FUNCTION_BLOCK TaskStoppingProbe EXTENDS TOF_Tasks.Task
VAR_INPUT
	//! <summary>Ordinary OnRunning result when no exception is injected.</summary>
	ProcessingResult : TOF_Tasks.TASK_PROCESSING_STATE := TOF_Tasks.TASK_PROCESSING_STATE.DONE;
	//! <summary>Throw from start preparation before RUNNING is entered.</summary>
	ThrowOnBeforeStart : BOOL;
	//! <summary>Throw when ordinary processing is called.</summary>
	ThrowOnRunning : BOOL;
	//! <summary>Throw once in stopping before advancing cleanup.</summary>
	ThrowOnFirstStopping : BOOL;
	//! <summary>Throw on every stopping call while enabled, before advancing cleanup.</summary>
	ThrowOnEveryStopping : BOOL;
	//! <summary>Throw from reset before descendant state is cleared.</summary>
	ThrowOnReset : BOOL;
	//! <summary>Injected exceptions throw again from GetMessage.</summary>
	ThrowOnGetMessage : BOOL;
	//! <summary>Throw a StandardException whose GetMessage result is empty.</summary>
	ThrowWithEmptyMessage : BOOL;
	//! <summary>Exercise the permitted Reset notification after termination.</summary>
	ResetOnAfterStop : BOOL;
END_VAR
VAR_OUTPUT
	//! <summary>Total ordinary processing calls across runs.</summary>
	RunningCalls : UINT;
	//! <summary>Total stopping-hook calls across runs, including interrupted calls.</summary>
	StoppingCalls : UINT;
	//! <summary>Successful stopping steps since the last Reset.</summary>
	CompletedCleanupSteps : UINT;
	//! <summary>Total notifications after STOPPED has been recorded.</summary>
	AfterStopCalls : UINT;
	//! <summary>Total accepted cancellation notifications.</summary>
	CancelNotifications : UINT;
END_VAR
VAR CONSTANT
	//! <summary>Successful cleanup steps required before release is safe.</summary>
	_CleanupSteps : UINT := 2;
END_VAR
VAR_STAT
	//! <summary>Class name shared by all instances of this function block.</summary>
	_ClassName : STRING := __POUNAME();
END_VAR
VAR
	_Resource : REFERENCE TO TaskStoppingResource;
	_StoppingExceptionRaised : BOOL;
END_VAR

{attribute 'monitoring' := 'call'}
PROPERTY ClassName : REFERENCE TO STRING
GET
ClassName REF= _ClassName;
END_GET
END_PROPERTY

(*!
<summary>Starts a fresh set of observation counts.</summary>
<description>
Call while the fixture is READY. Leaves configuration, cleanup progress and the borrowed resource binding intact.
</description>
*)
METHOD INTERNAL ClearObservations
RunningCalls := 0;
StoppingCalls := 0;
AfterStopCalls := 0;
CancelNotifications := 0;
END_METHOD

(*!
<summary>Borrows the test namespace.</summary>
*)
{attribute 'monitoring' := 'call'}
PROPERTY NamespaceName : REFERENCE TO STRING
GET
NamespaceName REF= CurrentNamespace.Name;
END_GET
END_PROPERTY

(*!
<summary>Counts finalization and optionally resets the stopped task.</summary>
<description>
Reset is invoked only after STOPPED and final diagnostics have been published.
</description>
*)
METHOD PROTECTED OnAfterStop
AfterStopCalls := AfterStopCalls + 1;

IF ResetOnAfterStop THEN
	Reset();
END_IF
END_METHOD

(*!
<summary>Optionally refuses start through an injected exception.</summary>
*)
METHOD PROTECTED OnBeforeStart
IF ThrowOnBeforeStart THEN
	raiseConfiguredFailure(message := "Start failure");
END_IF
END_METHOD

(*!
<summary>Counts accepted external cancellation notifications.</summary>
*)
METHOD PROTECTED OnCancelRequest
CancelNotifications := CancelNotifications + 1;
END_METHOD

(*!
<summary>Clears per-run cleanup progress without resetting observations or the dependency.</summary>
<description>
An injected exception refuses Reset before changing descendant state.
</description>
*)
METHOD PROTECTED OnReset
IF ThrowOnReset THEN
	raiseConfiguredFailure(message := "Reset failure");
END_IF

CompletedCleanupSteps := 0;
_StoppingExceptionRaised := FALSE;
END_METHOD

(*!
<summary>Returns the configured work result or injects a processing exception.</summary>
<description>
One call records one unit of work; no resource operations are driven here.
</description>
<param name="processingState">Configured result on normal return.</param>
<param name="stopReasonMessage">Receives diagnostic text for ERROR or ABORTED.</param>
*)
METHOD PROTECTED OnRunning
VAR_OUTPUT
	processingState : TOF_Tasks.TASK_PROCESSING_STATE;
END_VAR
VAR_IN_OUT
	stopReasonMessage : TOF_Core.ERROR_MESSAGE;
END_VAR
RunningCalls := RunningCalls + 1;

IF ThrowOnRunning THEN
	raiseConfiguredFailure(message := "Work failure");
END_IF

processingState := ProcessingResult;

IF processingState = TOF_Tasks.TASK_PROCESSING_STATE.ERROR
	OR_ELSE processingState = TOF_Tasks.TASK_PROCESSING_STATE.ABORTED
THEN
	stopReasonMessage := "Work result";
END_IF
END_METHOD

(*!
<summary>Finishes late acquisition and two cleanup steps before allowing release.</summary>
<description>
The configured exception can interrupt one or every call before progress. A later call resumes without
rerunning ordinary work once repeated injection is disabled.
</description>
<param name="readyToRelease">TRUE only after pending acquisition and cleanup have completed.</param>
*)
METHOD PROTECTED OnStopping
VAR_OUTPUT
	readyToRelease : BOOL;
END_VAR
StoppingCalls := StoppingCalls + 1;

IF ThrowOnFirstStopping AND_THEN NOT _StoppingExceptionRaised THEN
	_StoppingExceptionRaised := TRUE;
	raiseConfiguredFailure(message := "Stopping failure");
END_IF

IF ThrowOnEveryStopping THEN
	raiseConfiguredFailure(message := "Stopping failure");
END_IF

IF __ISVALIDREF(_Resource) AND_THEN NOT _Resource.FinishPendingAcquire() THEN
	RETURN;
END_IF

CompletedCleanupSteps := CompletedCleanupSteps + 1;
readyToRelease := CompletedCleanupSteps >= _CleanupSteps;
END_METHOD

(*!
<summary>Raises the configured synthetic exception.</summary>
<description>
Used only by test operations, never by FB lifecycle methods. A throwing or empty formatter exercises
diagnostic fallback.
</description>
<param name="message">Text copied into the injected exception.</param>
*)
METHOD PRIVATE raiseConfiguredFailure
VAR_INPUT
	message : WSTRING(255);
END_VAR
VAR
	failure : TOF_Core.StandardException;
	formattingFailure : ThrowingGetMessageException;
	emptyMessage : TOF_Core.ERROR_MESSAGE;
END_VAR
IF ThrowOnGetMessage THEN
	formattingFailure.Throw(
		sourceNamespaceName := NamespaceName,
		sourceClassName := ClassName,
		sourcePOUName := __POUNAME(),
		sourcePosition := __POSITION(),
		message := message
	);
ELSIF ThrowWithEmptyMessage THEN
	emptyMessage := TOF_Core.WideStrings.Empty;
	failure.Throw(
		sourceNamespaceName := NamespaceName,
		sourceClassName := ClassName,
		sourcePOUName := __POUNAME(),
		sourcePosition := __POSITION(),
		message := emptyMessage
	);
ELSE
	failure.Throw(
		sourceNamespaceName := NamespaceName,
		sourceClassName := ClassName,
		sourcePOUName := __POUNAME(),
		sourcePosition := __POSITION(),
		message := message
	);
END_IF
END_METHOD

(*!
<summary>Returns the explicitly injected borrowed resource manager.</summary>
<description>
Zero before binding; getter has no side effects and does not throw.
</description>
*)
{attribute 'monitoring' := 'call'}
PROPERTY ResourceManager : TOF_Core.IResourceManager
GET
IF __ISVALIDREF(_Resource) THEN
	ResourceManager := _Resource;
END_IF
END_GET
END_PROPERTY

(*!
<summary>Reports the concrete fixture size.</summary>
*)
{attribute 'monitoring' := 'call'}
PROPERTY SelfSize : ULINT
GET
SelfSize := XSIZEOF(THIS^);
END_GET
END_PROPERTY

(*!
<summary>Binds the manager owned by the scenario.</summary>
<description>
Call before Start and keep the referenced manager alive and unchanged throughout every run. Reset preserves
the binding.
</description>
<param name="resource">Live synthetic manager owned directly by the scenario.</param>
*)
METHOD INTERNAL SetResource
VAR_IN_OUT
	resource : TaskStoppingResource;
END_VAR
_Resource REF= resource;
END_METHOD

END_FUNCTION_BLOCK

// ---- Tests/Tasks/Stopping/TaskStoppingResource.TcPOU
(*
SPDX-FileCopyrightText: © 2026 Oleksandr Tiutyk <trofimich@gmail.com>
SPDX-License-Identifier: MIT
License: https://opensource.org/license/mit
*)

(*!
<summary>Provides delayed synthetic acquisition and release for Task stopping tests.</summary>
<description>
The scenario owns this manager and injects it into the task explicitly. Configure inputs before Start.
Operations have no hardware effects. A release exception intentionally leaves the synthetic resource held.
Observations are read-only to the scenario. ResetFixture clears them and the simulated state once the task is inactive.
</description>
*)

FUNCTION_BLOCK TaskStoppingResource EXTENDS TOF_Core.Object IMPLEMENTS TOF_Core.IResourceManager
VAR_INPUT
	//! <summary>Throw before acquisition is scheduled.</summary>
	ThrowOnStartAcquire : BOOL;
	//! <summary>Throw after the last acquisition step has marked the resource acquired.</summary>
	ThrowAfterAcquire : BOOL;
	//! <summary>Throw before release is scheduled, retaining the acquired resource.</summary>
	ThrowOnStartRelease : BOOL;
	//! <summary>Injected exceptions throw again when GetMessage is called.</summary>
	ThrowOnGetMessage : BOOL;
END_VAR
VAR_OUTPUT
	//! <summary>Total acquisition requests across runs.</summary>
	AcquireCalls : UINT;
	//! <summary>Total release requests across runs.</summary>
	ReleaseCalls : UINT;
	//! <summary>Completed steps in the current acquisition.</summary>
	AcquireProgress : UINT;
END_VAR
VAR CONSTANT
	//! <summary>Calls needed for a pending acquisition, allowing cancellation before its response.</summary>
	_AcquireSteps : UINT := 3;
	//! <summary>Calls needed after StartRelease to observe asynchronous completion.</summary>
	_ReleaseSteps : UINT := 2;
END_VAR
VAR_STAT
	//! <summary>Class name shared by all instances of this function block.</summary>
	_ClassName : STRING := __POUNAME();
END_VAR
VAR
	_Acquired : BOOL;
	_Acquiring : BOOL;
	_Releasing : BOOL;
	_ReleaseProgress : UINT;
END_VAR

{attribute 'monitoring' := 'call'}
PROPERTY ClassName : REFERENCE TO STRING
GET
ClassName REF= _ClassName;
END_GET
END_PROPERTY

(*!
<summary>Advances one pending synthetic operation.</summary>
<description>
No pending operation means no action. Acquisition failure may occur after ownership was obtained.
</description>
*)
METHOD Execute
IF _Acquiring THEN
	AcquireProgress := AcquireProgress + 1;

	IF AcquireProgress >= _AcquireSteps THEN
		_Acquiring := FALSE;
		_Acquired := TRUE;

		IF ThrowAfterAcquire THEN
			raiseConfiguredFailure(message := "Acquire failure");
		END_IF
	END_IF
ELSIF _Releasing THEN
	_ReleaseProgress := _ReleaseProgress + 1;

	IF _ReleaseProgress >= _ReleaseSteps THEN
		_Releasing := FALSE;
		_Acquired := FALSE;
	END_IF
END_IF
END_METHOD

(*!
<summary>Drains a late acquisition response without starting a new request.</summary>
<description>
Used by the injected task during OnStopping. A late acquired resource remains available for normal release.
</description>
*)
METHOD INTERNAL FinishPendingAcquire : BOOL
IF _Acquiring THEN
	Execute();
END_IF

FinishPendingAcquire := NOT _Acquiring;
END_METHOD

(*!
<summary>Returns the borrowed manager as a synthetic resource.</summary>
<description>
The caller must not delete it.
</description>
*)
METHOD GetResource : TOF_Core.IObject
GetResource := THIS^;
END_METHOD

(*!
<summary>Borrows the test namespace.</summary>
*)
{attribute 'monitoring' := 'call'}
PROPERTY NamespaceName : REFERENCE TO STRING
GET
NamespaceName REF= CurrentNamespace.Name;
END_GET
END_PROPERTY

(*!
<summary>Raises the configured synthetic exception.</summary>
<description>
Used only by test operations, never by FB lifecycle methods. The throwing formatter exercises diagnostic
fallback.
</description>
<param name="message">Text copied into the injected exception.</param>
*)
METHOD PRIVATE raiseConfiguredFailure
VAR_INPUT
	message : WSTRING(255);
END_VAR
VAR
	failure : TOF_Core.StandardException;
	formattingFailure : ThrowingGetMessageException;
END_VAR
IF ThrowOnGetMessage THEN
	formattingFailure.Throw(
		sourceNamespaceName := NamespaceName,
		sourceClassName := ClassName,
		sourcePOUName := __POUNAME(),
		sourcePosition := __POSITION(),
		message := message
	);
ELSE
	failure.Throw(
		sourceNamespaceName := NamespaceName,
		sourceClassName := ClassName,
		sourcePOUName := __POUNAME(),
		sourcePosition := __POSITION(),
		message := message
	);
END_IF
END_METHOD

(*!
<summary>Reports synthetic resource ownership.</summary>
<description>
Side-effect-free and non-throwing.
</description>
*)
{attribute 'monitoring' := 'call'}
PROPERTY ResourceAcquired : BOOL
GET
ResourceAcquired := _Acquired;
END_GET
END_PROPERTY

(*!
<summary>Reports the concrete fixture size.</summary>
*)
{attribute 'monitoring' := 'call'}
PROPERTY SelfSize : ULINT
GET
SelfSize := XSIZEOF(THIS^);
END_GET
END_PROPERTY

(*!
<summary>Restores idle synthetic state and clears all observations.</summary>
<description>
Call only when the driving task is inactive. Clears synthetic ownership even after an injected release failure.
Leaves fault configuration intact and does not perform physical release.
</description>
*)
METHOD INTERNAL ResetFixture
_Acquired := FALSE;
_Acquiring := FALSE;
_Releasing := FALSE;
_ReleaseProgress := 0;
AcquireProgress := 0;
AcquireCalls := 0;
ReleaseCalls := 0;
END_METHOD

(*!
<summary>Requests one delayed acquisition.</summary>
<description>
An injected early exception leaves no pending operation. An already acquired resource is retained.
</description>
*)
METHOD StartAcquire
AcquireCalls := AcquireCalls + 1;

IF ThrowOnStartAcquire THEN
	raiseConfiguredFailure(message := "Acquire failure");
END_IF

IF NOT _Acquired THEN
	AcquireProgress := 0;
	_Acquiring := TRUE;
END_IF
END_METHOD

(*!
<summary>Requests delayed release or throws the configured terminal failure.</summary>
<description>
The task must issue this once. A thrown request deliberately keeps ResourceAcquired TRUE.
</description>
*)
METHOD StartRelease
ReleaseCalls := ReleaseCalls + 1;

IF ThrowOnStartRelease THEN
	raiseConfiguredFailure(message := "Release failure");
END_IF

_ReleaseProgress := 0;
_Releasing := TRUE;
END_METHOD

END_FUNCTION_BLOCK

// ---- Tests/Tasks/Stopping/TaskStoppingScenarioTest.TcPOU
(*
SPDX-FileCopyrightText: © 2026 Oleksandr Tiutyk <trofimich@gmail.com>
SPDX-License-Identifier: MIT
License: https://opensource.org/license/mit
*)

(*!
<summary>Checks one cooperative stopping configuration of the production Task.</summary>
<description>
Owns persistent synthetic fixtures that perform no hardware work. One task drives the scenario using at most
one Execute per cycle. AfterTest drains remaining simulated work before preparing the fixtures for runner Reset.
</description>
*)

{attribute 'no_assign'}
{attribute 'no_explicit_call' := 'do not call this function block directly'}
FUNCTION_BLOCK TaskStoppingScenarioTest EXTENDS TOF_Testing.MultiCycleTest
VAR_STAT
	{attribute 'hide'}
	_ClassName : STRING := __POUNAME();
END_VAR
VAR CONSTANT
	//! <summary>Nominal call budget allowing acquisition, injected exceptions, cleanup and release.</summary>
	_MaxScenarioCalls : UDINT := 32;
	//! <summary>First observed acquisition step, before synthetic ownership can be acquired.</summary>
	_FirstAcquireStep : UINT := 1;
	//! <summary>Interrupt this many stopping calls before resuming in the repeated-fault case.</summary>
	_RepeatedStoppingFailures : UINT := 3;
	//! <summary>The probe must complete both successful cleanup steps before release or termination.</summary>
	_RequiredCleanupSteps : UINT := 2;
END_VAR
VAR
	_Scenario : TASK_STOPPING_TEST_SCENARIO;
	_Task : TaskStoppingProbe(name := "TaskStoppingProbe");
	_Resource : TaskStoppingResource;

	_ExpectedReason : TOF_Tasks.TASK_STOP_REASON;
	_ExpectedMessage : WSTRING(255);
	_ExpectedAcquireCalls : UINT;
	_ExpectedWorkCalls : UINT;
	_ExpectedReleaseCalls : UINT;
	_ExpectedStoppingCalls : UINT;
	_ExpectedCancelNotifications : UINT;

	_ObservedStopping : BOOL;
	_ObservedPendingRelease : BOOL;
	_CancelRequested : BOOL;
END_VAR

(*!
<summary>Stores the case and uses a cycle budget instead of a nominal duration.</summary>
<param name="name">Display name of the case.</param>
<param name="parent">Group that owns this case.</param>
<param name="scenario">Fault and observation configuration.</param>
*)
METHOD FB_init : BOOL
VAR_INPUT
	bInitRetains: BOOL; // TRUE: the retain variables are initialized (reset warm / reset cold)
	bInCopyCode: BOOL; // TRUE: the instance will be copied to the copy code afterward (online change)
	name : WSTRING;
	parent : TOF_Testing.ITestElement;
	scenario : TASK_STOPPING_TEST_SCENARIO;
END_VAR
_Scenario := scenario;
_Timeout := TOF_Core.Times.MIN_VALUE;
FB_init := TRUE;
END_METHOD

(*!
<summary>Prepares the chosen fixture before starting its observed run.</summary>
*)
METHOD PROTECTED BeforeTest
IF NOT _Task.State.Ready OR_ELSE _Resource.ResourceAcquired THEN
	RecordFailure(message := "The stopping fixture must begin READY without an acquired resource");
	RETURN;
END_IF

_Task.ClearObservations();
_ObservedStopping := FALSE;
_ObservedPendingRelease := FALSE;
_CancelRequested := FALSE;

configureScenario();

IF _Scenario = TASK_STOPPING_TEST_SCENARIO.START_FORMATTER_EXCEPTION THEN
	checkStartRefusal();

	IF Outcome = TOF_Testing.TEST_OUTCOME.FAILED THEN
		RETURN;
	END_IF
END_IF

IF NOT _Task.Start() THEN
	RecordFailure(message := "The prepared task must accept Start");
	RETURN;
END_IF

IF _Scenario = TASK_STOPPING_TEST_SCENARIO.CANCEL_BEFORE_ACQUIRE
	OR_ELSE _Scenario = TASK_STOPPING_TEST_SCENARIO.START_FORMATTER_EXCEPTION
THEN
	Assert.ThatBool(
		actual := _Task.Cancel(),
		message := "Cancellation before the first Execute must be accepted"
	).IsTrue();
END_IF
END_METHOD

(*!
<summary>Sets independent expected observations and applies the selected injections.</summary>
*)
METHOD PRIVATE configureScenario
_ExpectedReason := TOF_Tasks.TASK_STOP_REASON.WORK_DONE;
_ExpectedMessage := "";
_ExpectedAcquireCalls := 1;
_ExpectedWorkCalls := 1;
_ExpectedReleaseCalls := 1;
_ExpectedStoppingCalls := _RequiredCleanupSteps;
_ExpectedCancelNotifications := 0;

IF _Scenario <> TASK_STOPPING_TEST_SCENARIO.EMPTY_WORK_EXCEPTION_MESSAGE THEN
	_Task.SetResource(resource := _Resource);
END_IF

CASE _Scenario OF
	TASK_STOPPING_TEST_SCENARIO.WORK_ERROR:
		_Task.ProcessingResult := TOF_Tasks.TASK_PROCESSING_STATE.ERROR;
		_ExpectedReason := TOF_Tasks.TASK_STOP_REASON.FAILURE;
		_ExpectedMessage := "Work result";

	TASK_STOPPING_TEST_SCENARIO.WORK_ABORT:
		_Task.ProcessingResult := TOF_Tasks.TASK_PROCESSING_STATE.ABORTED;
		_ExpectedReason := TOF_Tasks.TASK_STOP_REASON.INTERNAL_ABORT;
		_ExpectedMessage := "Work result";

	TASK_STOPPING_TEST_SCENARIO.WORK_EXCEPTION,
	TASK_STOPPING_TEST_SCENARIO.WORK_FORMATTER_EXCEPTION,
	TASK_STOPPING_TEST_SCENARIO.FIRST_STOPPING_EXCEPTION,
	TASK_STOPPING_TEST_SCENARIO.EMPTY_WORK_EXCEPTION_MESSAGE:
		_Task.ThrowOnRunning := TRUE;
		_ExpectedReason := TOF_Tasks.TASK_STOP_REASON.FAILURE;
		_ExpectedMessage := "Work failure";

		CASE _Scenario OF
			TASK_STOPPING_TEST_SCENARIO.WORK_FORMATTER_EXCEPTION:
				_Task.ThrowOnGetMessage := TRUE;
				_ExpectedMessage := "Task 'TaskStoppingProbe' processing failed";

			TASK_STOPPING_TEST_SCENARIO.FIRST_STOPPING_EXCEPTION:
				_Task.ThrowOnFirstStopping := TRUE;
				_ExpectedStoppingCalls := _RequiredCleanupSteps + 1;

			TASK_STOPPING_TEST_SCENARIO.EMPTY_WORK_EXCEPTION_MESSAGE:
				_Task.ThrowWithEmptyMessage := TRUE;
				_ExpectedMessage := "Task 'TaskStoppingProbe' processing failed";
				_ExpectedAcquireCalls := 0;
				_ExpectedReleaseCalls := 0;
		END_CASE

	TASK_STOPPING_TEST_SCENARIO.REPEATED_STOPPING_EXCEPTIONS:
		_Task.ThrowOnEveryStopping := TRUE;
		_ExpectedStoppingCalls := _RequiredCleanupSteps + _RepeatedStoppingFailures;

	TASK_STOPPING_TEST_SCENARIO.CANCEL_DURING_ACQUIRE,
	TASK_STOPPING_TEST_SCENARIO.CANCEL_BEFORE_ACQUIRE,
	TASK_STOPPING_TEST_SCENARIO.START_FORMATTER_EXCEPTION:
		_ExpectedReason := TOF_Tasks.TASK_STOP_REASON.EXTERNAL_CANCEL;
		_ExpectedMessage := "Cancelled by external logic";
		_ExpectedWorkCalls := 0;
		_ExpectedCancelNotifications := 1;

		IF _Scenario = TASK_STOPPING_TEST_SCENARIO.CANCEL_DURING_ACQUIRE THEN
			_ExpectedStoppingCalls := _RequiredCleanupSteps + 1;
		ELSE
			_ExpectedAcquireCalls := 0;
			_ExpectedReleaseCalls := 0;
		END_IF

	TASK_STOPPING_TEST_SCENARIO.ACQUIRE_EXCEPTION_AFTER_OWNERSHIP:
		_Resource.ThrowAfterAcquire := TRUE;
		_Resource.ThrowOnGetMessage := TRUE;
		_ExpectedReason := TOF_Tasks.TASK_STOP_REASON.FAILURE;
		_ExpectedMessage := "Task 'TaskStoppingProbe' resource acquisition failed";
		_ExpectedWorkCalls := 0;

	TASK_STOPPING_TEST_SCENARIO.ACQUIRE_EXCEPTION_BEFORE_OWNERSHIP:
		_Resource.ThrowOnStartAcquire := TRUE;
		_ExpectedReason := TOF_Tasks.TASK_STOP_REASON.FAILURE;
		_ExpectedMessage := "Acquire failure";
		_ExpectedWorkCalls := 0;
		_ExpectedReleaseCalls := 0;

	TASK_STOPPING_TEST_SCENARIO.RELEASE_EXCEPTION:
		_Resource.ThrowOnStartRelease := TRUE;
		_Resource.ThrowOnGetMessage := TRUE;

	TASK_STOPPING_TEST_SCENARIO.RESET_IN_NOTIFICATION:
		_Task.ResetOnAfterStop := TRUE;
END_CASE
END_METHOD

(*!
<summary>Observes contained Start refusal before clearing the injection and retrying.</summary>
*)
METHOD PRIVATE checkStartRefusal
VAR
	refuseReason : TOF_Core.ERROR_MESSAGE;
END_VAR
_Task.ThrowOnBeforeStart := TRUE;
_Task.ThrowOnGetMessage := TRUE;

Assert.ThatBool(
	actual := _Task.Start(refuseReason => refuseReason),
	message := "The Start hook exception must refuse Start"
).IsFalse();
Assert.ThatBool(
	actual := _Task.State.Ready,
	message := "Refused Start must leave the task READY"
).IsTrue();
Assert.ThatUInt(
	actual := _Resource.AcquireCalls,
	message := "Refused Start must make no acquisition request"
).ToBe(expected := 0);
Assert.ThatWideString(
	actual := refuseReason,
	message := "Start must use the fixed formatter fallback"
).ToBe(expected := "Task start preparation failed");

_Task.ThrowOnBeforeStart := FALSE;
_Task.ThrowOnGetMessage := FALSE;
END_METHOD

(*!
<summary>Advances the observed task and reports its terminal observations.</summary>
<description>
After an injected terminal release failure, schedules an extra idle Execute to detect an unsolicited retry.
</description>
*)
METHOD PROTECTED ExecuteTest : TOF_Testing.TEST_CYCLE_RESULT
ExecuteTest := TOF_Testing.TEST_CYCLE_RESULT.DONE;

IF CycleCount > _MaxScenarioCalls THEN
	RecordFailure(message := "Task stopping exceeded its call budget");
	RETURN;
END_IF

IF _Task.State.Stopped AND_THEN _Scenario = TASK_STOPPING_TEST_SCENARIO.RELEASE_EXCEPTION THEN
	_Task.Execute();
	checkFinalObservations();
	checkFailedRelease();
	RETURN;
END_IF

_Task.Execute();

IF _Scenario = TASK_STOPPING_TEST_SCENARIO.CANCEL_DURING_ACQUIRE
	AND_THEN NOT _CancelRequested
	AND_THEN _Resource.AcquireProgress = _FirstAcquireStep
THEN
	_CancelRequested := _Task.Cancel();
	Assert.ThatBool(
		actual := _CancelRequested,
		message := "Cancelling pending acquisition must succeed"
	).IsTrue();
	Assert.ThatBool(
		actual := _Resource.ResourceAcquired,
		message := "Cancellation must precede the late acquire response"
	).IsFalse();
END_IF

IF _Task.State.Running THEN
	observeRunning();
	ExecuteTest := TOF_Testing.TEST_CYCLE_RESULT.BUSY;
	RETURN;
END_IF

checkFinalObservations();

CASE _Scenario OF
	TASK_STOPPING_TEST_SCENARIO.RELEASE_EXCEPTION:
		checkFailedRelease();
		ExecuteTest := TOF_Testing.TEST_CYCLE_RESULT.BUSY;

	TASK_STOPPING_TEST_SCENARIO.RESET_FORMATTER_EXCEPTION:
		IF Outcome <> TOF_Testing.TEST_OUTCOME.FAILED THEN
			checkResetRefusal();
		END_IF
END_CASE
END_METHOD

(*!
<summary>Checks the stopping transition and asynchronous release across calls.</summary>
*)
METHOD PRIVATE observeRunning
IF _Task.RunningSubstate.Stopping THEN
	Assert.ThatUInt(
		actual := _Resource.ReleaseCalls,
		message := "Release cannot start while stopping is incomplete"
	).ToBe(expected := 0);
	Assert.ThatBool(
		actual := _Task.OriginalStopReason.Value = _ExpectedReason,
		message := "Stopping must preserve the original reason"
	).IsTrue();

	IF NOT _ObservedStopping THEN
		_ObservedStopping := TRUE;
		checkFirstStoppingObservation();
	END_IF

	IF _Task.ThrowOnEveryStopping THEN
		Assert.ThatUInt(
			actual := _Task.CompletedCleanupSteps,
			message := "Interrupted stopping calls must not advance cleanup"
		).ToBe(expected := 0);

		IF _Task.StoppingCalls >= _RepeatedStoppingFailures THEN
			_Task.ThrowOnEveryStopping := FALSE;
		END_IF
	END_IF
ELSIF _Task.RunningSubstate.ResourceReleasing THEN
	Assert.ThatUInt(
		actual := _Task.CompletedCleanupSteps,
		message := "All cleanup steps must complete before release"
	).ToBe(expected := _RequiredCleanupSteps);
	Assert.ThatBool(
		actual := _Resource.ResourceAcquired,
		message := "Resource ownership must remain until release completes"
	).IsTrue();

	IF _Resource.ReleaseCalls = 1 THEN
		_ObservedPendingRelease := TRUE;
	END_IF
END_IF
END_METHOD

(*!
<summary>Distinguishes immediate normal stopping from stopping deferred by exceptions.</summary>
*)
METHOD PRIVATE checkFirstStoppingObservation
CASE _Scenario OF
	TASK_STOPPING_TEST_SCENARIO.WORK_EXCEPTION,
	TASK_STOPPING_TEST_SCENARIO.WORK_FORMATTER_EXCEPTION,
	TASK_STOPPING_TEST_SCENARIO.FIRST_STOPPING_EXCEPTION,
	TASK_STOPPING_TEST_SCENARIO.EMPTY_WORK_EXCEPTION_MESSAGE,
	TASK_STOPPING_TEST_SCENARIO.ACQUIRE_EXCEPTION_AFTER_OWNERSHIP,
	TASK_STOPPING_TEST_SCENARIO.ACQUIRE_EXCEPTION_BEFORE_OWNERSHIP,
	TASK_STOPPING_TEST_SCENARIO.CANCEL_DURING_ACQUIRE:
		Assert.ThatUInt(
			actual := _Task.StoppingCalls,
			message := "Stopping must wait for the next Execute"
		).ToBe(expected := 0);

	ELSE
		Assert.ThatUInt(
			actual := _Task.StoppingCalls,
			message := "The first stopping step must run in this Execute"
		).ToBe(expected := 1);
END_CASE
END_METHOD

(*!
<summary>Checks the finalization count, call counts and retained original and final results.</summary>
*)
METHOD PRIVATE checkFinalObservations
Assert.ThatBool(
	actual := _ObservedStopping,
	message := "The scenario must observe an active STOPPING phase"
).IsTrue();
Assert.ThatUInt(
	actual := _Task.RunningCalls,
	message := "Ordinary work must run only when expected"
).ToBe(expected := _ExpectedWorkCalls);
Assert.ThatUInt(
	actual := _Task.StoppingCalls,
	message := "Stopping calls must match the configured faults and cleanup"
).ToBe(expected := _ExpectedStoppingCalls);
Assert.ThatUInt(
	actual := _Task.AfterStopCalls,
	message := "Final notification must occur exactly once"
).ToBe(expected := 1);
Assert.ThatUInt(
	actual := _Task.CancelNotifications,
	message := "Accepted owner cancellation must notify exactly once"
).ToBe(expected := _ExpectedCancelNotifications);
Assert.ThatUInt(
	actual := _Resource.AcquireCalls,
	message := "Acquisition must be requested only when required"
).ToBe(expected := _ExpectedAcquireCalls);
Assert.ThatUInt(
	actual := _Resource.ReleaseCalls,
	message := "Release must be requested only when required"
).ToBe(expected := _ExpectedReleaseCalls);

IF _Scenario = TASK_STOPPING_TEST_SCENARIO.CANCEL_DURING_ACQUIRE THEN
	Assert.ThatUInt(
		actual := _Resource.AcquireProgress,
		message := "Cancelled acquisition must drain all three synthetic steps before releasing"
	).ToBe(expected := 3);
END_IF

IF _Scenario = TASK_STOPPING_TEST_SCENARIO.RESET_IN_NOTIFICATION THEN
	Assert.ThatBool(
		actual := _Task.State.Ready,
		message := "OnAfterStop Reset must leave the task READY without reentering work"
	).IsTrue();
	Assert.ThatUInt(
		actual := _Task.CompletedCleanupSteps,
		message := "Callback Reset must clear the stopping progress"
	).ToBe(expected := 0);
	Assert.ThatBool(
		actual := _Resource.ResourceAcquired,
		message := "Callback Reset must follow completed release"
	).IsFalse();
	Assert.ThatBool(
		actual := _ObservedPendingRelease,
		message := "Asynchronous release must be observable before the callback"
	).IsTrue();

	RETURN;
END_IF

Assert.ThatBool(actual := _Task.State.Stopped, message := "The task must have reached STOPPED").IsTrue();
Assert.ThatUInt(
	actual := _Task.CompletedCleanupSteps,
	message := "Both cleanup steps must complete before termination"
).ToBe(expected := _RequiredCleanupSteps);
Assert.ThatBool(
	actual := _Task.OriginalStopReason.Value = _ExpectedReason,
	message := "Cleanup must preserve the original reason"
).IsTrue();
Assert.ThatWideString(
	actual := _Task.OriginalStopReason.Message,
	message := "Cleanup must preserve the original diagnostic"
).ToBe(expected := _ExpectedMessage);

IF _Scenario = TASK_STOPPING_TEST_SCENARIO.RELEASE_EXCEPTION THEN
	RETURN;
END_IF

Assert.ThatBool(
	actual := _Task.FinalStopReason.Value = _ExpectedReason,
	message := "After successful cleanup the final reason must match"
).IsTrue();
Assert.ThatBool(
	actual := _Resource.ResourceAcquired,
	message := "Successful cleanup must leave the resource released"
).IsFalse();
Assert.ThatBool(
	actual := _ObservedPendingRelease = (_ExpectedReleaseCalls = 1),
	message := "Only a requested asynchronous release must remain pending"
).IsTrue();

IF _ExpectedMessage <> "" THEN
	Assert.ThatWideString(
		actual := _Task.FinalStopReason.Message,
		message := "Final diagnostic must retain the original text"
	).ToBe(expected := _ExpectedMessage);
END_IF
END_METHOD

(*!
<summary>Checks terminal release failure and preserves the work result.</summary>
*)
METHOD PRIVATE checkFailedRelease
Assert.ThatBool(
	actual := _Task.State.Stopped AND_THEN _Task.FinalStopReason.Failure,
	message := "Terminal release failure must leave STOPPED with FAILURE"
).IsTrue();
Assert.ThatBool(
	actual := _Task.OriginalStopReason.WorkDone,
	message := "Failed release must preserve the original successful work result"
).IsTrue();
Assert.ThatWideString(
	actual := _Task.FinalStopReason.Message,
	message := "Failed release formatter must use the named fallback"
).ToBe(expected := "Task 'TaskStoppingProbe' release failed");
Assert.ThatBool(
	actual := _Resource.ResourceAcquired,
	message := "Failed release must leave the synthetic resource held"
).IsTrue();
Assert.ThatUInt(
	actual := _Resource.ReleaseCalls,
	message := "Failed release must not be retried"
).ToBe(expected := 1);
Assert.ThatUInt(
	actual := _Task.AfterStopCalls,
	message := "Failed release must not repeat final notification"
).ToBe(expected := 1);
END_METHOD

(*!
<summary>Verifies fixed diagnostics and retries Reset after removing the injected fault.</summary>
*)
METHOD PRIVATE checkResetRefusal
VAR
	refuseReason : TOF_Core.ERROR_MESSAGE;
END_VAR
_Task.ThrowOnReset := TRUE;
_Task.ThrowOnGetMessage := TRUE;

Assert.ThatBool(
	actual := _Task.Reset(refuseReason => refuseReason),
	message := "A resetting hook exception must refuse Reset"
).IsFalse();
Assert.ThatBool(actual := _Task.State.Stopped, message := "Refused Reset must preserve STOPPED").IsTrue();
Assert.ThatWideString(
	actual := refuseReason,
	message := "Reset must use the fixed formatter fallback"
).ToBe(expected := "Task reset failed");

_Task.ThrowOnReset := FALSE;
_Task.ThrowOnGetMessage := FALSE;
Assert.ThatBool(
	actual := _Task.Reset(),
	message := "Reset must succeed after removing the injected failure"
).IsTrue();
Assert.ThatBool(
	actual := _Task.State.Ready,
	message := "Successful Reset must prepare the task for reuse"
).IsTrue();
END_METHOD

(*!
<summary>Clears injections and drains simulated work before publishing the outcome.</summary>
<description>
The bounded drain runs only on synchronous synthetic fixtures. If the task remains active or refuses Reset,
does not clear the simulated resource state. Clears a held test resource after the terminal result was observed.
</description>
*)
METHOD PROTECTED AfterTest
VAR
	i : UDINT;
END_VAR
_Task.ProcessingResult := TOF_Tasks.TASK_PROCESSING_STATE.DONE;
_Task.ThrowOnBeforeStart := FALSE;
_Task.ThrowOnRunning := FALSE;
_Task.ThrowOnFirstStopping := FALSE;
_Task.ThrowOnEveryStopping := FALSE;
_Task.ThrowOnReset := FALSE;
_Task.ThrowOnGetMessage := FALSE;
_Task.ThrowWithEmptyMessage := FALSE;
_Task.ResetOnAfterStop := FALSE;
_Resource.ThrowOnStartAcquire := FALSE;
_Resource.ThrowAfterAcquire := FALSE;
_Resource.ThrowOnStartRelease := FALSE;
_Resource.ThrowOnGetMessage := FALSE;

__TRY
	IF _Task.State.Running THEN
		IF NOT _Task.OriginalStopReason.ExternalCancel AND_THEN NOT _Task.RunningSubstate.ResourceReleasing THEN
			_Task.Cancel();
		END_IF

		FOR i := 1 TO _MaxScenarioCalls DO
			IF NOT _Task.State.Running THEN
				EXIT;
			END_IF

			_Task.Execute();
		END_FOR
	END_IF
__CATCH
	reportCleanupFailure(message := "An exception interrupted synthetic stopping or release");
__ENDTRY

IF _Task.State.Running THEN
	reportCleanupFailure(message := "Synthetic cleanup left the task RUNNING");
	RETURN;
END_IF

IF _Task.State.Stopped THEN
	IF NOT _Task.Reset() THEN
		reportCleanupFailure(message := "Stopped probe refused cleanup Reset");
		RETURN;
	END_IF
END_IF

IF NOT _Task.State.Ready THEN
	reportCleanupFailure(message := "The probe must return to READY after cleanup");
	RETURN;
END_IF

_Resource.ResetFixture();
END_METHOD

(*!
<summary>Reports cleanup failures without overwriting a recorded outcome.</summary>
<param name="message">Cleanup diagnostic copied to the test or ADS log.</param>
*)
METHOD PRIVATE reportCleanupFailure
VAR_IN_OUT CONSTANT
	message : TOF_Core.ERROR_MESSAGE;
END_VAR
VAR
	logText : STRING(255);
END_VAR
IF Outcome = TOF_Testing.TEST_OUTCOME.FAILED THEN
	logText := TO_STRING(TOF_Core.WideStrings.ConcatFit255(Name, " cleanup: ", TO_WSTRING(message)));
	Tc2_System.ADSLOGSTR(
		msgCtrlMask := Tc2_System.Global_Variables.ADSLOG_MSGTYPE_ERROR,
		msgFmtStr := '%s',
		strArg := logText
	);
ELSE
	RecordFailure(message := message);
END_IF
END_METHOD

//! <summary>Borrows the concrete class name. Callers must not modify it.</summary>
{attribute 'monitoring' := 'call'}
PROPERTY ClassName : REFERENCE TO STRING
GET
ClassName REF= _ClassName;
END_GET
END_PROPERTY

//! <summary>Borrows the compiler-initialized namespace name. Callers must not modify it.</summary>
{attribute 'monitoring' := 'call'}
PROPERTY NamespaceName : REFERENCE TO STRING
GET
NamespaceName REF= CurrentNamespace.Name;
END_GET
END_PROPERTY

//! <summary>Reports the concrete instance size in bytes.</summary>
{attribute 'monitoring' := 'call'}
PROPERTY SelfSize : ULINT
GET
SelfSize := XSIZEOF(THIS^);
END_GET
END_PROPERTY

END_FUNCTION_BLOCK

// ---- Tests/Core/ObjectLifetimeTestGroup.TcPOU
(*
SPDX-FileCopyrightText: © 2026 Oleksandr Tiutyk <trofimich@gmail.com>
SPDX-License-Identifier: MIT
License: https://opensource.org/license/mit
*)

(*!
<summary>Groups the four object lifetime cases.</summary>
<description>
Owns the independent child instances and their fixed registration array. Use from one PLC task at a stable address.
</description>
*)

{attribute 'no_assign'}
{attribute 'no_explicit_call' := 'do not call this function block directly'}
FUNCTION_BLOCK ObjectLifetimeTestGroup EXTENDS TOF_Testing.TestGroup<4>
VAR_STAT
	{attribute 'hide'}
	_ClassName : STRING := __POUNAME();
END_VAR
VAR
	_TypedDeletion : DynamicObjectDisposalTest(
		name := "DeleteTypedPointer",
		parent := THIS^,
		releaseThroughInterface := FALSE
	);
	_InterfaceDeletion : DynamicObjectDisposalTest(
		name := "DeleteThroughIObject",
		parent := THIS^,
		releaseThroughInterface := TRUE
	);
	_Address : ObjectInterfaceAddressTest(name := "GetInstanceAddress", parent := THIS^);
	_StaticRefusal : StaticObjectReleaseRefusalTest(name := "RefuseStaticObjectRelease", parent := THIS^);

	_Children : ARRAY [0.._ChildCount - 1] OF TOF_Testing.ITestElement :=
	[
		_TypedDeletion,
		_InterfaceDeletion,
		_Address,
		_StaticRefusal
	];
END_VAR

//! <summary>Borrows the fixed child array. Callers must not modify it.</summary>
{attribute 'monitoring' := 'call'}
PROPERTY Children : REFERENCE TO ARRAY [0.._ChildCount - 1] OF TOF_Testing.ITestElement
GET
Children REF= _Children;
END_GET
END_PROPERTY

//! <summary>Borrows the concrete class name. Callers must not modify it.</summary>
{attribute 'monitoring' := 'call'}
PROPERTY ClassName : REFERENCE TO STRING
GET
ClassName REF= _ClassName;
END_GET
END_PROPERTY

//! <summary>Borrows the compiler-initialized namespace name. Callers must not modify it.</summary>
{attribute 'monitoring' := 'call'}
PROPERTY NamespaceName : REFERENCE TO STRING
GET
NamespaceName REF= CurrentNamespace.Name;
END_GET
END_PROPERTY

//! <summary>Reports the concrete instance size in bytes.</summary>
{attribute 'monitoring' := 'call'}
PROPERTY SelfSize : ULINT
GET
SelfSize := XSIZEOF(THIS^);
END_GET
END_PROPERTY

END_FUNCTION_BLOCK

// ---- Tests/Core/DynamicObjectDisposalTest.TcPOU
(*
SPDX-FileCopyrightText: © 2026 Oleksandr Tiutyk <trofimich@gmail.com>
SPDX-License-Identifier: MIT
License: https://opensource.org/license/mit
*)

(*!
<summary>Verifies concrete destruction through typed deletion or IObject.</summary>
<description>
Owns one dynamic probe at a time. The exit counter remains live through deletion. The test uses each
ownership path once per run and executes in one PLC task. AfterTest deletes only a probe still owned by this case.
</description>
*)

{attribute 'no_assign'}
{attribute 'no_explicit_call' := 'do not call this function block directly'}
FUNCTION_BLOCK DynamicObjectDisposalTest EXTENDS TOF_Testing.SingleCycleTest
VAR_STAT
	{attribute 'hide'}
	_ClassName : STRING := __POUNAME();
END_VAR
VAR
	_ReleaseThroughInterface : BOOL;
	_OwnedProbe : POINTER TO ObjectExitProbe;
	_ExitCount : UDINT;
END_VAR

(*!
<summary>Selects the disposal route for this case.</summary>
<param name="name">Display name of this case.</param>
<param name="parent">Group that owns this case.</param>
<param name="releaseThroughInterface">TRUE selects Memory.TryReleaseDynamicObject. FALSE selects typed __DELETE.</param>
*)
METHOD FB_init : BOOL
VAR_INPUT
	bInitRetains: BOOL; // TRUE: the retain variables are initialized (reset warm / reset cold)
	bInCopyCode: BOOL; // TRUE: the instance will be copied to the copy code afterward (online change)
	name : WSTRING;
	parent : TOF_Testing.ITestElement;
	releaseThroughInterface : BOOL;
END_VAR
_ReleaseThroughInterface := releaseThroughInterface;
FB_init := TRUE;
END_METHOD

(*!
<summary>Allocates a fresh probe and verifies its concrete exit count.</summary>
<description>
A failed allocation follows the fatal allocation boundary. The exit counter is cleared before each allocation.
</description>
*)
METHOD PROTECTED ExecuteTest
_ExitCount := 0;
_OwnedProbe := __NEW(ObjectExitProbe);

IF _OwnedProbe = 0 THEN
	TOF_Core.DynamicMemoryManager.RaiseAllocationFailure();
	RETURN;
END_IF

_OwnedProbe^.ObserveExit(counter := _ExitCount);

IF _ReleaseThroughInterface THEN
	checkInterfaceRelease();
ELSE
	deleteOwnedProbe();
	Assert.ThatUDInt(
		actual := _ExitCount,
		message := "Typed deletion must call the concrete FB_exit once"
	).ToBe(expected := 1);
END_IF
END_METHOD

(*!
<summary>Checks interface address resolution, destruction and repeat release of the cleared interface.</summary>
<description>
After passing the interface to the release helper, does not dereference or re-delete the former allocation.
A repeated call is allowed only after confirmed success with a null interface.
</description>
*)
METHOD PRIVATE checkInterfaceRelease
VAR
	instance : TOF_Core.IObject;
	released : BOOL;
END_VAR
instance := _OwnedProbe^;
Assert.ThatBool(
	actual := TOF_Core.Memory.GetAddressFromInterface(interfaceInstance := instance) = _OwnedProbe,
	message := "The dynamic interface must resolve to the complete probe address"
).IsTrue();

// Give up the typed alias before an operation that can leave the object partially destroyed.
_OwnedProbe := 0;
released := TOF_Core.Memory.TryReleaseDynamicObject(instance := instance);
Assert.ThatBool(actual := released, message := "Live dynamic probe release must succeed").IsTrue();
Assert.ThatBool(actual := instance = 0, message := "Release must clear the passed interface").IsTrue();
Assert.ThatUDInt(
	actual := _ExitCount,
	message := "Interface release must call the concrete FB_exit once"
).ToBe(expected := 1);

IF NOT released OR_ELSE instance <> 0 THEN
	RETURN;
END_IF

released := TOF_Core.Memory.TryReleaseDynamicObject(instance := instance);
Assert.ThatBool(actual := released, message := "Repeated release of the cleared interface must return FALSE").IsFalse();
Assert.ThatBool(actual := instance = 0, message := "Repeated release must leave the interface clear").IsTrue();
Assert.ThatUDInt(
	actual := _ExitCount,
	message := "Repeated release must not call FB_exit again"
).ToBe(expected := 1);
END_METHOD

(*!
<summary>Cleans up a probe still owned by the case after an interrupted preparation.</summary>
*)
METHOD PROTECTED AfterTest
IF _OwnedProbe <> 0 THEN
	deleteOwnedProbe();
END_IF
END_METHOD

(*!
<summary>Deletes the live probe through its exact type and clears the ownership field before deletion.</summary>
<description>
Call only when this case still owns the live allocation. The probe implements a non-throwing exit.
</description>
*)
METHOD PRIVATE deleteOwnedProbe
VAR
	probe : POINTER TO ObjectExitProbe;
END_VAR
probe := _OwnedProbe;
_OwnedProbe := 0;
__DELETE(probe);
END_METHOD

//! <summary>Borrows the concrete class name. Callers must not modify it.</summary>
{attribute 'monitoring' := 'call'}
PROPERTY ClassName : REFERENCE TO STRING
GET
ClassName REF= _ClassName;
END_GET
END_PROPERTY

//! <summary>Borrows the compiler-initialized namespace name. Callers must not modify it.</summary>
{attribute 'monitoring' := 'call'}
PROPERTY NamespaceName : REFERENCE TO STRING
GET
NamespaceName REF= CurrentNamespace.Name;
END_GET
END_PROPERTY

//! <summary>Reports the concrete instance size in bytes.</summary>
{attribute 'monitoring' := 'call'}
PROPERTY SelfSize : ULINT
GET
SelfSize := XSIZEOF(THIS^);
END_GET
END_PROPERTY

END_FUNCTION_BLOCK

// ---- Tests/Core/ObjectExitProbe.TcPOU
(*
SPDX-FileCopyrightText: © 2026 Oleksandr Tiutyk <trofimich@gmail.com>
SPDX-License-Identifier: MIT
License: https://opensource.org/license/mit
*)

{attribute 'enable_dynamic_creation'}
{attribute 'no_explicit_call' := 'Direct call is not allowed'}
FUNCTION_BLOCK ObjectExitProbe EXTENDS TOF_Core.Object
VAR_STAT
	//! <summary>Class name shared by all instances of this function block.</summary>
	_ClassName : STRING := __POUNAME();
END_VAR
VAR
	_ExitCounter : REFERENCE TO UDINT;
END_VAR

(*!
<summary>The counter must remain alive until this instance is deleted.</summary>
*)

METHOD ObserveExit
VAR_IN_OUT
	counter : UDINT;
END_VAR
_ExitCounter REF= counter;
END_METHOD

METHOD FB_exit : BOOL
VAR_INPUT
	bInCopyCode : BOOL;
END_VAR
IF __ISVALIDREF(_ExitCounter) THEN
	_ExitCounter := _ExitCounter + 1;
END_IF
END_METHOD

PROPERTY ClassName : REFERENCE TO STRING
GET
ClassName REF= _ClassName;
END_GET
END_PROPERTY

PROPERTY NamespaceName : REFERENCE TO STRING
GET
NamespaceName REF= CurrentNamespace.Name;
END_GET
END_PROPERTY

PROPERTY SelfSize : ULINT
GET
SelfSize := XSIZEOF(THIS^);
END_GET
END_PROPERTY

END_FUNCTION_BLOCK

// ---- Tests/Core/ObjectInterfaceAddressTest.TcPOU
(*
SPDX-FileCopyrightText: © 2026 Oleksandr Tiutyk <trofimich@gmail.com>
SPDX-License-Identifier: MIT
License: https://opensource.org/license/mit
*)

(*!
<summary>Checks interface-to-instance address conversion for a static object and for null.</summary>
<description>
Uses an owned static fixture. The converted address is borrowed and compared only in the calling task.
</description>
*)

{attribute 'no_assign'}
{attribute 'no_explicit_call' := 'do not call this function block directly'}
FUNCTION_BLOCK ObjectInterfaceAddressTest EXTENDS TOF_Testing.SingleCycleTest
VAR_STAT
	{attribute 'hide'}
	_ClassName : STRING := __POUNAME();
END_VAR
VAR
	_Probe : ObjectExitProbe;
END_VAR

(*!
<summary>Converts the live static interface, then checks that a null input does not reuse the address.</summary>
*)
METHOD PROTECTED ExecuteTest
VAR
	instance : TOF_Core.IObject;
END_VAR
instance := _Probe;
Assert.ThatBool(
	actual := TOF_Core.Memory.GetAddressFromInterface(interfaceInstance := instance) = ADR(_Probe),
	message := "The static interface must resolve to the complete probe address"
).IsTrue();

instance := 0;
Assert.ThatBool(
	actual := TOF_Core.Memory.GetAddressFromInterface(interfaceInstance := instance) = 0,
	message := "A null interface must return zero after a successful conversion"
).IsTrue();
END_METHOD

//! <summary>Borrows the concrete class name. Callers must not modify it.</summary>
{attribute 'monitoring' := 'call'}
PROPERTY ClassName : REFERENCE TO STRING
GET
ClassName REF= _ClassName;
END_GET
END_PROPERTY

//! <summary>Borrows the compiler-initialized namespace name. Callers must not modify it.</summary>
{attribute 'monitoring' := 'call'}
PROPERTY NamespaceName : REFERENCE TO STRING
GET
NamespaceName REF= CurrentNamespace.Name;
END_GET
END_PROPERTY

//! <summary>Reports the concrete instance size in bytes.</summary>
{attribute 'monitoring' := 'call'}
PROPERTY SelfSize : ULINT
GET
SelfSize := XSIZEOF(THIS^);
END_GET
END_PROPERTY

END_FUNCTION_BLOCK

// ---- Tests/Core/StaticObjectReleaseRefusalTest.TcPOU
(*
SPDX-FileCopyrightText: © 2026 Oleksandr Tiutyk <trofimich@gmail.com>
SPDX-License-Identifier: MIT
License: https://opensource.org/license/mit
*)

(*!
<summary>Checks that the dynamic release helper refuses to destroy a static object.</summary>
<description>
Owns a static probe and a persistent exit counter. Each run binds and clears the counter before making the
release request. The test executes in one PLC task and keeps the probe at a stable address.
</description>
*)

{attribute 'no_assign'}
{attribute 'no_explicit_call' := 'do not call this function block directly'}
FUNCTION_BLOCK StaticObjectReleaseRefusalTest EXTENDS TOF_Testing.SingleCycleTest
VAR_STAT
	{attribute 'hide'}
	_ClassName : STRING := __POUNAME();
END_VAR
VAR
	_Probe : ObjectExitProbe;
	_ExitCount : UDINT;
END_VAR

(*!
<summary>Checks refusal, preserved interface identity and absence of a concrete exit call.</summary>
*)
METHOD PROTECTED ExecuteTest
VAR
	instance : TOF_Core.IObject;
	originalInstance : TOF_Core.IObject;
	released : BOOL;
END_VAR
_ExitCount := 0;
_Probe.ObserveExit(counter := _ExitCount);
instance := _Probe;
originalInstance := instance;
released := TOF_Core.Memory.TryReleaseDynamicObject(instance := instance);

Assert.ThatBool(actual := released, message := "Static instance release must be refused").IsFalse();
Assert.ThatBool(
	actual := instance = originalInstance,
	message := "Refusal must preserve the original static interface"
).IsTrue();
Assert.ThatUDInt(
	actual := _ExitCount,
	message := "Refusal must not call the static probe FB_exit"
).ToBe(expected := 0);
END_METHOD

//! <summary>Borrows the concrete class name. Callers must not modify it.</summary>
{attribute 'monitoring' := 'call'}
PROPERTY ClassName : REFERENCE TO STRING
GET
ClassName REF= _ClassName;
END_GET
END_PROPERTY

//! <summary>Borrows the compiler-initialized namespace name. Callers must not modify it.</summary>
{attribute 'monitoring' := 'call'}
PROPERTY NamespaceName : REFERENCE TO STRING
GET
NamespaceName REF= CurrentNamespace.Name;
END_GET
END_PROPERTY

//! <summary>Reports the concrete instance size in bytes.</summary>
{attribute 'monitoring' := 'call'}
PROPERTY SelfSize : ULINT
GET
SelfSize := XSIZEOF(THIS^);
END_GET
END_PROPERTY

END_FUNCTION_BLOCK

// ---- Tests/Core/GenericValueTestGroup.TcPOU
(*
SPDX-FileCopyrightText: c 2026 Oleksandr Tiutyk <trofimich@gmail.com>
SPDX-License-Identifier: MIT
License: https://opensource.org/license/mit
*)

(*!
<summary>Groups generic storage, ordering, conversion and runtime type diagnostics.</summary>
<description>
Owns the independent child instances and their fixed registration array. Use from one PLC task at a stable address.
</description>
*)

{attribute 'no_assign'}
{attribute 'no_explicit_call' := 'do not call this function block directly'}
FUNCTION_BLOCK GenericValueTestGroup EXTENDS TOF_Testing.TestGroup<8>
VAR_STAT
	{attribute 'hide'}
	_ClassName : STRING := __POUNAME();
END_VAR
VAR
	_LongStrings : GenericLongStringOrderingTest(name := "LongStringOrdering", parent := THIS^);
	_StringPrefixes : GenericStringPrefixOrderingTest(name := "StringPrefixAndEncodingOrder", parent := THIS^);
	_NaNs : GenericNaNOrderingTest(name := "NaNOrdering", parent := THIS^);
	_MixedNumericPrecision : GenericMixedNumericPrecisionTest(name := "MixedNumericPrecision", parent := THIS^);
	_ConversionPairs : GenericConversionPairsTest(name := "SupportedConversionPairs", parent := THIS^);
	_TypeClassFormatting : SystemTypeClassFormattingTest(name := "SystemTypeClassFormatting", parent := THIS^);
	_TypeClassDiagnostics : SystemTypeClassDiagnosticsTest(name := "TypeClassDiagnostics", parent := THIS^);
	_BorrowedWrites : GenericBorrowedWritesTest(name := "ChangesCompatibleValues", parent := THIS^);

	_Children : ARRAY [0.._ChildCount - 1] OF TOF_Testing.ITestElement :=
	[
		_LongStrings,
		_StringPrefixes,
		_NaNs,
		_MixedNumericPrecision,
		_ConversionPairs,
		_TypeClassFormatting,
		_TypeClassDiagnostics,
		_BorrowedWrites
	];
END_VAR

//! <summary>Borrows the fixed child array. Callers must not modify it.</summary>
{attribute 'monitoring' := 'call'}
PROPERTY Children : REFERENCE TO ARRAY [0.._ChildCount - 1] OF TOF_Testing.ITestElement
GET
Children REF= _Children;
END_GET
END_PROPERTY

//! <summary>Borrows the concrete class name. Callers must not modify it.</summary>
{attribute 'monitoring' := 'call'}
PROPERTY ClassName : REFERENCE TO STRING
GET
ClassName REF= _ClassName;
END_GET
END_PROPERTY

//! <summary>Borrows the compiler-initialized namespace name. Callers must not modify it.</summary>
{attribute 'monitoring' := 'call'}
PROPERTY NamespaceName : REFERENCE TO STRING
GET
NamespaceName REF= CurrentNamespace.Name;
END_GET
END_PROPERTY

//! <summary>Reports the concrete instance size in bytes.</summary>
{attribute 'monitoring' := 'call'}
PROPERTY SelfSize : ULINT
GET
SelfSize := XSIZEOF(THIS^);
END_GET
END_PROPERTY

END_FUNCTION_BLOCK

// ---- Tests/Core/GenericLongStringOrderingTest.TcPOU
(*
SPDX-FileCopyrightText: c 2026 Oleksandr Tiutyk <trofimich@gmail.com>
SPDX-License-Identifier: MIT
License: https://opensource.org/license/mit
*)

(*!
<summary>Compares strings that differ after character 255.</summary>
<description>
Uses run-local fixtures and references that are used only within the executing PLC task.
The runner binds assertions to the instance address. Keep the instance at that address for its run.
</description>
*)

{attribute 'no_assign'}
{attribute 'no_explicit_call' := 'do not call this function block directly'}
FUNCTION_BLOCK GenericLongStringOrderingTest EXTENDS TOF_Testing.SingleCycleTest
VAR_STAT
	{attribute 'hide'}
	_ClassName : STRING := __POUNAME();
END_VAR

(*!
<summary>Checks ordering after a 299-character common prefix in both string encodings.</summary>
<description>
Includes narrow, wide and mixed operands, reverse order and equality beyond 255 characters.
Both 300-character fixtures contain ASCII and explicitly terminate their buffers at offset 300.
</description>
*)
METHOD PROTECTED ExecuteTest
VAR
	narrowFirst : STRING(300);
	narrowSecond : STRING(300);
	wideFirst : WSTRING(300);
	wideSecond : WSTRING(300);
	wideFirstData : POINTER TO WORD;
	wideSecondData : POINTER TO WORD;
	first : TOF_Core.GENERIC_VALUE;
	second : TOF_Core.GENERIC_VALUE;
	i : INT;
END_VAR
wideFirstData := ADR(wideFirst);
wideSecondData := ADR(wideSecond);

// SA0175: Construct and explicitly terminate 300-byte ASCII operands.
{analysis -175}
FOR i := 0 TO 299 DO
	narrowFirst[i] := BYTE#16#61;
	narrowSecond[i] := BYTE#16#61;
	wideFirstData[i] := WORD#16#61;
	wideSecondData[i] := WORD#16#61;
END_FOR

narrowSecond[299] := BYTE#16#62;
narrowFirst[300] := TO_BYTE(TOF_Core.UnsignedInt8.MIN_VALUE);
narrowSecond[300] := TO_BYTE(TOF_Core.UnsignedInt8.MIN_VALUE);
{analysis +175}
wideSecondData[299] := WORD#16#62;
wideFirstData[300] := TO_WORD(TOF_Core.UnsignedInt16.MIN_VALUE);
wideSecondData[300] := TO_WORD(TOF_Core.UnsignedInt16.MIN_VALUE);
first := TOF_Core.GenericValueFactory.FromStringReference(value := narrowFirst);
second := TOF_Core.GenericValueFactory.FromStringReference(value := narrowSecond);
Assert.ThatBool(
	actual := first.CompareTo(otherValue := second) = TOF_Core.COMPARISON_RESULT.FIRST_LESS_THAN_SECOND,
	message := "Narrow ordering must include characters after position 255"
).IsTrue();

first := TOF_Core.GenericValueFactory.FromWStringReference(value := wideFirst);
second := TOF_Core.GenericValueFactory.FromWStringReference(value := wideSecond);
Assert.ThatBool(
	actual := first.CompareTo(otherValue := second) = TOF_Core.COMPARISON_RESULT.FIRST_LESS_THAN_SECOND,
	message := "Wide ordering must include characters after position 255"
).IsTrue();

first := TOF_Core.GenericValueFactory.FromStringReference(value := narrowFirst);
Assert.ThatBool(
	actual := first.CompareTo(otherValue := second) = TOF_Core.COMPARISON_RESULT.FIRST_LESS_THAN_SECOND,
	message := "Mixed ordering must include the complete narrow and wide strings"
).IsTrue();
Assert.ThatBool(
	actual := second.CompareTo(otherValue := first) = TOF_Core.COMPARISON_RESULT.FIRST_GREATER_THAN_SECOND,
	message := "Reversing mixed operands must reverse the result"
).IsTrue();

second := TOF_Core.GenericValueFactory.FromWStringReference(value := wideFirst);
Assert.ThatBool(
	actual := first.CompareTo(otherValue := second) = TOF_Core.COMPARISON_RESULT.FIRST_EQUAL_TO_SECOND,
	message := "Equal long strings must compare equal across encodings"
).IsTrue();
END_METHOD

//! <summary>Borrows the concrete class name. Callers must not modify it.</summary>
{attribute 'monitoring' := 'call'}
PROPERTY ClassName : REFERENCE TO STRING
GET
ClassName REF= _ClassName;
END_GET
END_PROPERTY

//! <summary>Borrows the compiler-initialized namespace name. Callers must not modify it.</summary>
{attribute 'monitoring' := 'call'}
PROPERTY NamespaceName : REFERENCE TO STRING
GET
NamespaceName REF= CurrentNamespace.Name;
END_GET
END_PROPERTY

//! <summary>Reports the concrete instance size in bytes.</summary>
{attribute 'monitoring' := 'call'}
PROPERTY SelfSize : ULINT
GET
SelfSize := XSIZEOF(THIS^);
END_GET
END_PROPERTY

END_FUNCTION_BLOCK

// ---- Tests/Core/GenericStringPrefixOrderingTest.TcPOU
(*
SPDX-FileCopyrightText: c 2026 Oleksandr Tiutyk <trofimich@gmail.com>
SPDX-License-Identifier: MIT
License: https://opensource.org/license/mit
*)

(*!
<summary>Checks mixed-encoding prefixes and unsigned code units.</summary>
<description>
Uses run-local fixtures and references that are used only within the executing PLC task.
The runner binds assertions to the instance address. Keep the instance at that address for its run.
</description>
*)

{attribute 'no_assign'}
{attribute 'no_explicit_call' := 'do not call this function block directly'}
FUNCTION_BLOCK GenericStringPrefixOrderingTest EXTENDS TOF_Testing.SingleCycleTest
VAR_STAT
	{attribute 'hide'}
	_ClassName : STRING := __POUNAME();
END_VAR

(*!
<summary>Checks terminators, prefixes and unsigned Latin-1 code units in mixed string comparisons.</summary>
<description>
Uses terminated buffers and confirms both operand directions without encoding conversions.
The FF fixture deliberately writes one Latin-1 byte rather than a UTF-8 sequence.
</description>
*)
METHOD PROTECTED ExecuteTest
VAR
	narrow : STRING(2);
	wide : WSTRING(2);
	wideData : POINTER TO WORD;
	first : TOF_Core.GENERIC_VALUE;
	second : TOF_Core.GENERIC_VALUE;
END_VAR
first := TOF_Core.GenericValueFactory.FromStringReference(value := narrow);
second := TOF_Core.GenericValueFactory.FromWStringReference(value := wide);
Assert.ThatBool(
	actual := first.CompareTo(otherValue := second) = TOF_Core.COMPARISON_RESULT.FIRST_EQUAL_TO_SECOND,
	message := "Empty strings must compare equal across encodings"
).IsTrue();

narrow := 'a';
wide := "ab";
first := TOF_Core.GenericValueFactory.FromStringReference(value := narrow);
second := TOF_Core.GenericValueFactory.FromWStringReference(value := wide);
Assert.ThatBool(
	actual := first.CompareTo(otherValue := second) = TOF_Core.COMPARISON_RESULT.FIRST_LESS_THAN_SECOND,
	message := "A prefix must precede a longer string"
).IsTrue();
Assert.ThatBool(
	actual := second.CompareTo(otherValue := first) = TOF_Core.COMPARISON_RESULT.FIRST_GREATER_THAN_SECOND,
	message := "A longer string must follow its prefix"
).IsTrue();

// SA0175: The test requires one Latin-1 FF code unit, not a UTF-8 sequence, followed by a terminator.
{analysis -175}
narrow[0] := BYTE#16#FF;
narrow[1] := BYTE#0;
{analysis +175}
wideData := ADR(wide);
wideData[0] := WORD#16#FF;
wideData[1] := WORD#0;
first := TOF_Core.GenericValueFactory.FromStringReference(value := narrow);
second := TOF_Core.GenericValueFactory.FromWStringReference(value := wide);
Assert.ThatBool(
	actual := first.CompareTo(otherValue := second) = TOF_Core.COMPARISON_RESULT.FIRST_EQUAL_TO_SECOND,
	message := "Latin-1 FF must widen to code unit 00FF"
).IsTrue();

wideData[0] := WORD#16#100;
Assert.ThatBool(
	actual := first.CompareTo(otherValue := second) = TOF_Core.COMPARISON_RESULT.FIRST_LESS_THAN_SECOND,
	message := "Latin-1 FF must precede UTF-16 0100"
).IsTrue();
END_METHOD

//! <summary>Borrows the concrete class name. Callers must not modify it.</summary>
{attribute 'monitoring' := 'call'}
PROPERTY ClassName : REFERENCE TO STRING
GET
ClassName REF= _ClassName;
END_GET
END_PROPERTY

//! <summary>Borrows the compiler-initialized namespace name. Callers must not modify it.</summary>
{attribute 'monitoring' := 'call'}
PROPERTY NamespaceName : REFERENCE TO STRING
GET
NamespaceName REF= CurrentNamespace.Name;
END_GET
END_PROPERTY

//! <summary>Reports the concrete instance size in bytes.</summary>
{attribute 'monitoring' := 'call'}
PROPERTY SelfSize : ULINT
GET
SelfSize := XSIZEOF(THIS^);
END_GET
END_PROPERTY

END_FUNCTION_BLOCK

// ---- Tests/Core/GenericNaNOrderingTest.TcPOU
(*
SPDX-FileCopyrightText: c 2026 Oleksandr Tiutyk <trofimich@gmail.com>
SPDX-License-Identifier: MIT
License: https://opensource.org/license/mit
*)

(*!
<summary>Checks NaN ordering across widths and number categories.</summary>
<description>
Uses run-local fixtures and references that are used only within the executing PLC task.
The runner binds assertions to the instance address. Keep the instance at that address for its run.
</description>
*)

{attribute 'no_assign'}
{attribute 'no_explicit_call' := 'do not call this function block directly'}
FUNCTION_BLOCK GenericNaNOrderingTest EXTENDS TOF_Testing.SingleCycleTest
VAR_STAT
	{attribute 'hide'}
	_ClassName : STRING := __POUNAME();
END_VAR

(*!
<summary>Checks that every NaN precedes non-NaN numbers and NaN encodings compare equal.</summary>
<description>
Constructs quiet and signaling NaN bit patterns without floating-point arithmetic. Includes both widths,
integers, negative infinity, reverse order and ordinary finite ordering.
</description>
*)
METHOD PROTECTED ExecuteTest
VAR
	narrowNaN : TOF_Core.REAL_UNION;
	wideNaN : TOF_Core.LREAL_UNION;
	negativeInfinity : TOF_Core.LREAL_UNION;
	integer : LINT;
	first : TOF_Core.GENERIC_VALUE;
	second : TOF_Core.GENERIC_VALUE;
END_VAR
narrowNaN.Raw := UDINT#16#7F800001;
wideNaN.Raw := ULINT#16#FFF8000000000011;
negativeInfinity.Raw := ULINT#16#FFF0000000000000;
first := TOF_Core.GenericValueFactory.FromRealReference(value := narrowNaN.Value);
second := TOF_Core.GenericValueFactory.FromLRealReference(value := wideNaN.Value);
Assert.ThatBool(
	actual := first.CompareTo(otherValue := second) = TOF_Core.COMPARISON_RESULT.FIRST_EQUAL_TO_SECOND,
	message := "Signaling REAL NaN and quiet LREAL NaN must compare equal"
).IsTrue();
Assert.ThatBool(
	actual := second.CompareTo(otherValue := first) = TOF_Core.COMPARISON_RESULT.FIRST_EQUAL_TO_SECOND,
	message := "NaN equality must be symmetric across widths"
).IsTrue();

second := TOF_Core.GenericValueFactory.FromLRealReference(value := negativeInfinity.Value);
Assert.ThatBool(
	actual := first.CompareTo(otherValue := second) = TOF_Core.COMPARISON_RESULT.FIRST_LESS_THAN_SECOND,
	message := "NaN must precede negative infinity"
).IsTrue();
Assert.ThatBool(
	actual := second.CompareTo(otherValue := first) = TOF_Core.COMPARISON_RESULT.FIRST_GREATER_THAN_SECOND,
	message := "Negative infinity must follow NaN"
).IsTrue();

second := TOF_Core.GenericValueFactory.FromLIntReference(value := integer);
Assert.ThatBool(
	actual := first.CompareTo(otherValue := second) = TOF_Core.COMPARISON_RESULT.FIRST_LESS_THAN_SECOND,
	message := "NaN must precede an integer"
).IsTrue();
Assert.ThatBool(
	actual := second.CompareTo(otherValue := first) = TOF_Core.COMPARISON_RESULT.FIRST_GREATER_THAN_SECOND,
	message := "An integer must follow NaN"
).IsTrue();

wideNaN.Raw := ULINT#16#7FF0000000000001;
first := TOF_Core.GenericValueFactory.FromLRealReference(value := wideNaN.Value);
Assert.ThatBool(
	actual := first.CompareTo(otherValue := second) = TOF_Core.COMPARISON_RESULT.FIRST_LESS_THAN_SECOND,
	message := "Signaling LREAL NaN must be classified before conversion or comparison"
).IsTrue();

wideNaN.Value := LREAL#1.0;
Assert.ThatBool(
	actual := first.CompareTo(otherValue := second) = TOF_Core.COMPARISON_RESULT.FIRST_GREATER_THAN_SECOND,
	message := "Ordinary finite numeric ordering must remain unchanged"
).IsTrue();
END_METHOD

//! <summary>Borrows the concrete class name. Callers must not modify it.</summary>
{attribute 'monitoring' := 'call'}
PROPERTY ClassName : REFERENCE TO STRING
GET
ClassName REF= _ClassName;
END_GET
END_PROPERTY

//! <summary>Borrows the compiler-initialized namespace name. Callers must not modify it.</summary>
{attribute 'monitoring' := 'call'}
PROPERTY NamespaceName : REFERENCE TO STRING
GET
NamespaceName REF= CurrentNamespace.Name;
END_GET
END_PROPERTY

//! <summary>Reports the concrete instance size in bytes.</summary>
{attribute 'monitoring' := 'call'}
PROPERTY SelfSize : ULINT
GET
SelfSize := XSIZEOF(THIS^);
END_GET
END_PROPERTY

END_FUNCTION_BLOCK

// ---- Tests/Core/GenericMixedNumericPrecisionTest.TcPOU
(*
SPDX-FileCopyrightText: c 2026 Oleksandr Tiutyk <trofimich@gmail.com>
SPDX-License-Identifier: MIT
License: https://opensource.org/license/mit
*)

(*!
<summary>Checks integer-to-floating comparisons at exact representation boundaries.</summary>
<description>
Uses run-local fixtures and references that are used only within the executing PLC task.
The runner binds assertions to the instance address. Keep the instance at that address for its run.
</description>
*)

{attribute 'no_assign'}
{attribute 'no_explicit_call' := 'do not call this function block directly'}
FUNCTION_BLOCK GenericMixedNumericPrecisionTest EXTENDS TOF_Testing.SingleCycleTest
VAR_STAT
	{attribute 'hide'}
	_ClassName : STRING := __POUNAME();
END_VAR

(*!
<summary>Checks exact integer-to-floating ordering at precision, range and fractional boundaries.</summary>
<description>
Uses independent expected directions for both operand orders. Values around 2^53 reproduce the transitivity
defect caused by converting integers to LREAL. Raw patterns cover signed zero, subnormal and infinite values.
</description>
*)
METHOD PROTECTED ExecuteTest
VAR
	signedInteger : LINT;
	unsignedInteger : ULINT;
	floatingValue : LREAL;
	narrowReal : REAL;
	realBits : TOF_Core.LREAL_UNION;
	integerValue : TOF_Core.GENERIC_VALUE;
	realValue : TOF_Core.GENERIC_VALUE;
END_VAR
integerValue := TOF_Core.GenericValueFactory.FromLIntReference(value := signedInteger);
realValue := TOF_Core.GenericValueFactory.FromLRealReference(value := floatingValue);
floatingValue := LREAL#9007199254740992.0;
signedInteger := LINT#9007199254740993;
assertOrder(
	first := integerValue,
	second := realValue,
	expected := TOF_Core.COMPARISON_RESULT.FIRST_GREATER_THAN_SECOND,
	scenario := "Integer one above 2^53"
);
signedInteger := LINT#9007199254740992;
assertOrder(
	first := integerValue,
	second := realValue,
	expected := TOF_Core.COMPARISON_RESULT.FIRST_EQUAL_TO_SECOND,
	scenario := "Integer equal to 2^53"
);
signedInteger := LINT#9007199254740991;
assertOrder(
	first := integerValue,
	second := realValue,
	expected := TOF_Core.COMPARISON_RESULT.FIRST_LESS_THAN_SECOND,
	scenario := "Integer one below 2^53"
);

floatingValue := LREAL#-9007199254740992.0;
signedInteger := LINT#-9007199254740993;
assertOrder(
	first := integerValue,
	second := realValue,
	expected := TOF_Core.COMPARISON_RESULT.FIRST_LESS_THAN_SECOND,
	scenario := "Integer below negative 2^53"
);
signedInteger := LINT#-9007199254740991;
assertOrder(
	first := integerValue,
	second := realValue,
	expected := TOF_Core.COMPARISON_RESULT.FIRST_GREATER_THAN_SECOND,
	scenario := "Integer above negative 2^53"
);

floatingValue := LREAL#9223372036854775808.0;
signedInteger := TOF_Core.SignedInt64.MAX_VALUE;
assertOrder(
	first := integerValue,
	second := realValue,
	expected := TOF_Core.COMPARISON_RESULT.FIRST_LESS_THAN_SECOND,
	scenario := "LINT maximum against 2^63"
);
floatingValue := LREAL#-9223372036854775808.0;
signedInteger := TOF_Core.SignedInt64.MIN_VALUE;
assertOrder(
	first := integerValue,
	second := realValue,
	expected := TOF_Core.COMPARISON_RESULT.FIRST_EQUAL_TO_SECOND,
	scenario := "LINT minimum against negative 2^63"
);

integerValue := TOF_Core.GenericValueFactory.FromULIntReference(value := unsignedInteger);
floatingValue := LREAL#18446744073709551616.0;
unsignedInteger := TOF_Core.UnsignedInt64.MAX_VALUE;
assertOrder(
	first := integerValue,
	second := realValue,
	expected := TOF_Core.COMPARISON_RESULT.FIRST_LESS_THAN_SECOND,
	scenario := "ULINT maximum against 2^64"
);
floatingValue := LREAL#9223372036854775808.0;
unsignedInteger := ULINT#9223372036854775809;
assertOrder(
	first := integerValue,
	second := realValue,
	expected := TOF_Core.COMPARISON_RESULT.FIRST_GREATER_THAN_SECOND,
	scenario := "Unsigned integer one above 2^63"
);

integerValue := TOF_Core.GenericValueFactory.FromLIntReference(value := signedInteger);
signedInteger := -1;
floatingValue := LREAL#-0.5;
assertOrder(
	first := integerValue,
	second := realValue,
	expected := TOF_Core.COMPARISON_RESULT.FIRST_LESS_THAN_SECOND,
	scenario := "Negative integer against negative half"
);
signedInteger := 0;
assertOrder(
	first := integerValue,
	second := realValue,
	expected := TOF_Core.COMPARISON_RESULT.FIRST_GREATER_THAN_SECOND,
	scenario := "Zero against negative half"
);
floatingValue := LREAL#0.5;
assertOrder(
	first := integerValue,
	second := realValue,
	expected := TOF_Core.COMPARISON_RESULT.FIRST_LESS_THAN_SECOND,
	scenario := "Zero against positive half"
);
signedInteger := 1;
assertOrder(
	first := integerValue,
	second := realValue,
	expected := TOF_Core.COMPARISON_RESULT.FIRST_GREATER_THAN_SECOND,
	scenario := "Positive integer against positive half"
);
signedInteger := 42;
floatingValue := LREAL#42.0;
assertOrder(
	first := integerValue,
	second := realValue,
	expected := TOF_Core.COMPARISON_RESULT.FIRST_EQUAL_TO_SECOND,
	scenario := "Equal positive integral operands"
);
floatingValue := LREAL#42.5;
assertOrder(
	first := integerValue,
	second := realValue,
	expected := TOF_Core.COMPARISON_RESULT.FIRST_LESS_THAN_SECOND,
	scenario := "Positive integer against a larger fraction"
);
floatingValue := LREAL#-42.5;
signedInteger := -42;
assertOrder(
	first := integerValue,
	second := realValue,
	expected := TOF_Core.COMPARISON_RESULT.FIRST_GREATER_THAN_SECOND,
	scenario := "Negative integer against a smaller fraction"
);

realValue := TOF_Core.GenericValueFactory.FromLRealReference(value := realBits.Value);
signedInteger := 0;
realBits.Raw := ULINT#16#8000000000000000;
assertOrder(
	first := integerValue,
	second := realValue,
	expected := TOF_Core.COMPARISON_RESULT.FIRST_EQUAL_TO_SECOND,
	scenario := "Integer zero against negative floating zero"
);
realBits.Raw := ULINT#1;
assertOrder(
	first := integerValue,
	second := realValue,
	expected := TOF_Core.COMPARISON_RESULT.FIRST_LESS_THAN_SECOND,
	scenario := "Zero against the smallest positive LREAL subnormal"
);
realBits.Raw := ULINT#16#7FF0000000000000;
assertOrder(
	first := integerValue,
	second := realValue,
	expected := TOF_Core.COMPARISON_RESULT.FIRST_LESS_THAN_SECOND,
	scenario := "Zero against positive infinity"
);
realBits.Raw := ULINT#16#FFF0000000000000;
assertOrder(
	first := integerValue,
	second := realValue,
	expected := TOF_Core.COMPARISON_RESULT.FIRST_GREATER_THAN_SECOND,
	scenario := "Zero against negative infinity"
);

narrowReal := REAL#16777216.0;
signedInteger := LINT#16777217;
realValue := TOF_Core.GenericValueFactory.FromRealReference(value := narrowReal);
assertOrder(
	first := integerValue,
	second := realValue,
	expected := TOF_Core.COMPARISON_RESULT.FIRST_GREATER_THAN_SECOND,
	scenario := "Integer above the REAL precision limit"
);
END_METHOD

(*!
<summary>Checks a numeric comparison and its reverse against an independently supplied expected direction.</summary>
<description>Borrows both descriptors for assertions; no payload mutation or ownership transfer occurs.</description>
<param name="first">First numeric descriptor.</param>
<param name="second">Second numeric descriptor.</param>
<param name="expected">Expected comparison of first with second.</param>
<param name="scenario">Boundary name included in assertion failures.</param>
*)
METHOD PRIVATE assertOrder
VAR_INPUT
	first : TOF_Core.GENERIC_VALUE;
	second : TOF_Core.GENERIC_VALUE;
	expected : TOF_Core.COMPARISON_RESULT;
	scenario : WSTRING(255);
END_VAR
VAR
	reversedExpected : TOF_Core.COMPARISON_RESULT;
END_VAR
CASE expected OF
	TOF_Core.COMPARISON_RESULT.FIRST_LESS_THAN_SECOND:
		reversedExpected := TOF_Core.COMPARISON_RESULT.FIRST_GREATER_THAN_SECOND;
	TOF_Core.COMPARISON_RESULT.FIRST_EQUAL_TO_SECOND:
		reversedExpected := TOF_Core.COMPARISON_RESULT.FIRST_EQUAL_TO_SECOND;
	TOF_Core.COMPARISON_RESULT.FIRST_GREATER_THAN_SECOND:
		reversedExpected := TOF_Core.COMPARISON_RESULT.FIRST_LESS_THAN_SECOND;
END_CASE

Assert.ThatSInt(
	actual := TO_SINT(first.CompareTo(otherValue := second)),
	message := Tc2_Utilities.WCONCAT(STR1 := "Integer first: ", STR2 := scenario)
).ToBe(expected := TO_SINT(expected));
Assert.ThatSInt(
	actual := TO_SINT(second.CompareTo(otherValue := first)),
	message := Tc2_Utilities.WCONCAT(STR1 := "Float first: ", STR2 := scenario)
).ToBe(expected := TO_SINT(reversedExpected));
END_METHOD

//! <summary>Borrows the concrete class name. Callers must not modify it.</summary>
{attribute 'monitoring' := 'call'}
PROPERTY ClassName : REFERENCE TO STRING
GET
ClassName REF= _ClassName;
END_GET
END_PROPERTY

//! <summary>Borrows the compiler-initialized namespace name. Callers must not modify it.</summary>
{attribute 'monitoring' := 'call'}
PROPERTY NamespaceName : REFERENCE TO STRING
GET
NamespaceName REF= CurrentNamespace.Name;
END_GET
END_PROPERTY

//! <summary>Reports the concrete instance size in bytes.</summary>
{attribute 'monitoring' := 'call'}
PROPERTY SelfSize : ULINT
GET
SelfSize := XSIZEOF(THIS^);
END_GET
END_PROPERTY

END_FUNCTION_BLOCK

// ---- Tests/Core/GenericConversionPairsTest.TcPOU
(*
SPDX-FileCopyrightText: c 2026 Oleksandr Tiutyk <trofimich@gmail.com>
SPDX-License-Identifier: MIT
License: https://opensource.org/license/mit
*)

(*!
<summary>Checks generic conversion availability and typed accessor behavior.</summary>
<description>
Uses run-local fixtures and references that are used only within the executing PLC task.
The runner binds assertions to the instance address. Keep the instance at that address for its run.
</description>
*)

{attribute 'no_assign'}
{attribute 'no_explicit_call' := 'do not call this function block directly'}
FUNCTION_BLOCK GenericConversionPairsTest EXTENDS TOF_Testing.SingleCycleTest
VAR_STAT
	{attribute 'hide'}
	_ClassName : STRING := __POUNAME();
END_VAR

(*!
<summary>Checks supported pairs without dereferencing payload and keeps range checks in the accessors.</summary>
<description>
Uses non-owning descriptors over passive storage for category queries and typed numeric descriptors for
selected conversions. Query-only descriptors are never read through typed accessors. Covers former false
positives, numeric-to-calendar false negatives, asymmetric date pairs and unsupported identity targets.
A deliberate range error checks the accessor separately.
</description>
*)
METHOD PROTECTED ExecuteTest
VAR
	value : TOF_Core.GENERIC_VALUE;
	queryStorage : LWORD;
	duration : TIME := T#1MS;
	integer : LINT := 0;
	convertedDate : DATE;
	exceptionCode : __SYSTEM.ExceptionCode;
	caughtException : TOF_Core.IException;
	conversionException : TOF_Core.IGenericConversionNotSupportedException;
END_VAR
value := TOF_Core.GenericValueFactory.FromParts(
	genericTypeClass := TOF_Core.GENERIC_TYPE_CLASS.OBJECT,
	address := ADR(queryStorage),
	size := XSIZEOF(queryStorage),
	memoryManagementBehavior :=
		TOF_Core.GENERIC_MEMORY_MANAGEMENT_BEHAVIOR.STORE_ORIGINAL_REFERENCE_AND_NOT_OWNS_MEMORY
);
Assert.ThatBool(
	actual := value.IsConvertibleTo(targetTypeClass := TOF_Core.GENERIC_TYPE_CLASS.STRING_16),
	message := "OBJECT has no text accessor conversion"
).IsFalse();

value := TOF_Core.GenericValueFactory.FromParts(
	genericTypeClass := TOF_Core.GENERIC_TYPE_CLASS.REAL_64,
	address := ADR(queryStorage),
	size := XSIZEOF(queryStorage),
	memoryManagementBehavior :=
		TOF_Core.GENERIC_MEMORY_MANAGEMENT_BEHAVIOR.STORE_ORIGINAL_REFERENCE_AND_NOT_OWNS_MEMORY
);
Assert.ThatBool(
	actual := value.IsConvertibleTo(targetTypeClass := TOF_Core.GENERIC_TYPE_CLASS.INT_32),
	message := "Floating-point to integer is not an accessor conversion"
).IsFalse();
Assert.ThatBool(
	actual := value.IsConvertibleTo(targetTypeClass := TOF_Core.GENERIC_TYPE_CLASS.REAL_32),
	message := "A query inspects the category without interpreting the borrowed payload"
).IsTrue();

value := TOF_Core.GenericValueFactory.FromParts(
	genericTypeClass := TOF_Core.GENERIC_TYPE_CLASS.DATE_AND_TIME_64,
	address := ADR(queryStorage),
	size := XSIZEOF(queryStorage),
	memoryManagementBehavior :=
		TOF_Core.GENERIC_MEMORY_MANAGEMENT_BEHAVIOR.STORE_ORIGINAL_REFERENCE_AND_NOT_OWNS_MEMORY
);
Assert.ThatBool(
	actual := value.IsConvertibleTo(targetTypeClass := TOF_Core.GENERIC_TYPE_CLASS.DATE_32),
	message := "AsDate does not provide an LDT input branch"
).IsFalse();
Assert.ThatBool(
	actual := value.IsConvertibleTo(targetTypeClass := TOF_Core.GENERIC_TYPE_CLASS.DATE_64),
	message := "AsLDate supports LDT input"
).IsTrue();

value := TOF_Core.GenericValueFactory.FromParts(
	genericTypeClass := TOF_Core.GENERIC_TYPE_CLASS.POINTER_TO,
	address := ADR(queryStorage),
	size := XSIZEOF(queryStorage),
	memoryManagementBehavior :=
		TOF_Core.GENERIC_MEMORY_MANAGEMENT_BEHAVIOR.STORE_ORIGINAL_REFERENCE_AND_NOT_OWNS_MEMORY
);
Assert.ThatBool(
	actual := value.IsConvertibleTo(targetTypeClass := TOF_Core.GENERIC_TYPE_CLASS.POINTER_TO),
	message := "A pointer identity tag has no As* accessor"
).IsFalse();
value := TOF_Core.GenericValueFactory.FromParts(
	genericTypeClass := TOF_Core.GENERIC_TYPE_CLASS.USER_DEFINED,
	address := ADR(queryStorage),
	size := XSIZEOF(queryStorage),
	memoryManagementBehavior :=
		TOF_Core.GENERIC_MEMORY_MANAGEMENT_BEHAVIOR.STORE_ORIGINAL_REFERENCE_AND_NOT_OWNS_MEMORY
);
Assert.ThatBool(
	actual := value.IsConvertibleTo(targetTypeClass := TOF_Core.GENERIC_TYPE_CLASS.USER_DEFINED),
	message := "A user-defined identity tag has no As* accessor"
).IsFalse();

value := TOF_Core.GenericValueFactory.FromLIntReference(value := integer);
Assert.ThatBool(
	actual := value.IsConvertibleTo(targetTypeClass := TOF_Core.GENERIC_TYPE_CLASS.DATE_32),
	message := "Integer seconds have a DATE conversion branch"
).IsTrue();
convertedDate := value.AsDate();
Assert.ThatDate(
	actual := convertedDate,
	message := "Zero seconds must convert to the epoch"
).ToBe(expected := DATE#1970-01-01);
integer := TOF_Core.SignedInt64.MAX_VALUE;
Assert.ThatBool(
	actual := value.IsConvertibleTo(targetTypeClass := TOF_Core.GENERIC_TYPE_CLASS.DATE_32),
	message := "A pair query must not become a value range check"
).IsTrue();

// Catch the deliberate out-of-range conversion to verify that the accessor rejects it.
__TRY
	convertedDate := value.AsDate(allowTypeCastWithDataLoss := TRUE);
__CATCH(exceptionCode)
	caughtException := TOF_Core.ExceptionManager.GetLastException(
		exceptionCode := exceptionCode,
		catchPointNamespaceName := NamespaceName,
		catchPointPOUName := __POUNAME(),
		catchPointPosition := __POSITION()
	);
__ENDTRY

Assert.ThatBool(
	actual := __QUERYINTERFACE(caughtException, conversionException),
	message := "An out-of-range integer must fail AsDate even when truncating time of day is allowed"
).IsTrue();

value := TOF_Core.GenericValueFactory.FromTimeReference(value := duration);
Assert.ThatBool(
	actual := value.IsConvertibleTo(targetTypeClass := TOF_Core.GENERIC_TYPE_CLASS.DATE_AND_TIME_64),
	message := "TIME has a conversion to LDT"
).IsTrue();
Assert.ThatLongDateTime(
	actual := value.AsLDateAndTime(),
	message := "TIME must add one millisecond to the epoch"
).ToBe(expected := LDT#1970-01-01-00:00:00.001);
END_METHOD

//! <summary>Borrows the concrete class name. Callers must not modify it.</summary>
{attribute 'monitoring' := 'call'}
PROPERTY ClassName : REFERENCE TO STRING
GET
ClassName REF= _ClassName;
END_GET
END_PROPERTY

//! <summary>Borrows the compiler-initialized namespace name. Callers must not modify it.</summary>
{attribute 'monitoring' := 'call'}
PROPERTY NamespaceName : REFERENCE TO STRING
GET
NamespaceName REF= CurrentNamespace.Name;
END_GET
END_PROPERTY

//! <summary>Reports the concrete instance size in bytes.</summary>
{attribute 'monitoring' := 'call'}
PROPERTY SelfSize : ULINT
GET
SelfSize := XSIZEOF(THIS^);
END_GET
END_PROPERTY

END_FUNCTION_BLOCK

// ---- Tests/Core/SystemTypeClassFormattingTest.TcPOU
(*
SPDX-FileCopyrightText: c 2026 Oleksandr Tiutyk <trofimich@gmail.com>
SPDX-License-Identifier: MIT
License: https://opensource.org/license/mit
*)

(*!
<summary>Checks symbolic runtime names and unknown code formatting.</summary>
<description>
Uses run-local fixtures and references that are used only within the executing PLC task.
The runner binds assertions to the instance address. Keep the instance at that address for its run.
</description>
*)

{attribute 'no_assign'}
{attribute 'no_explicit_call' := 'do not call this function block directly'}
FUNCTION_BLOCK SystemTypeClassFormattingTest EXTENDS TOF_Testing.SingleCycleTest
VAR_STAT
	{attribute 'hide'}
	_ClassName : STRING := __POUNAME();
END_VAR

(*!
<summary>Checks symbolic runtime names in both encodings and lossless formatting of unknown codes.</summary>
<description>
Covers reference, pointer, text, sentinel and Build 4026 extended categories. Injects an unknown raw DWORD
to exercise the fallback without requiring an enum conversion outside the declared values.
</description>
*)
METHOD PROTECTED ExecuteTest
VAR
	typeClasses : ARRAY [0..7] OF __SYSTEM.TYPE_CLASS := [
		__SYSTEM.TYPE_CLASS.TYPE_BOOL,
		__SYSTEM.TYPE_CLASS.TYPE_REFERENCE,
		__SYSTEM.TYPE_CLASS.TYPE_POINTER,
		__SYSTEM.TYPE_CLASS.TYPE_STRING,
		__SYSTEM.TYPE_CLASS.TYPE_WSTRING,
		__SYSTEM.TYPE_CLASS.TYPE_NONE,
		__SYSTEM.TYPE_CLASS.TYPE_ANYSTRING,
		__SYSTEM.TYPE_CLASS.TYPE_LTIMEOFDAY
	];
	expectedNames : ARRAY [0..7] OF STRING(80) := [
		'TYPE_BOOL', 'TYPE_REFERENCE', 'TYPE_POINTER', 'TYPE_STRING',
		'TYPE_WSTRING', 'TYPE_NONE', 'TYPE_ANYSTRING', 'TYPE_LTIMEOFDAY'
	];
	typeClass : __SYSTEM.TYPE_CLASS;
	unknownCode : DWORD := DWORD#16#FFFFFFFF;
	narrowName : STRING(80);
	caseName : WSTRING(80);
	wideName : WSTRING(80);

	i : INT;
END_VAR
FOR i := 0 TO 7 DO
	narrowName := TOF_Core.SystemTypeClassConvertor.ToString(typeClass := typeClasses[i]);
	wideName := TOF_Core.SystemTypeClassConvertor.ToWideString(typeClass := typeClasses[i]);
	caseName := TO_WSTRING(expectedNames[i]);
	Assert.ThatBool(
		actual := narrowName = expectedNames[i],
		message := Tc2_Utilities.WCONCAT(STR1 := "Incorrect STRING name for ", STR2 := caseName)
	).IsTrue();
	Assert.ThatBool(
		actual := wideName = caseName,
		message := Tc2_Utilities.WCONCAT(STR1 := "Incorrect WSTRING name for ", STR2 := caseName)
	).IsTrue();
END_FOR

// Preserve all 32 bits of an unknown runtime code, including the unsigned high bit.
Tc2_System.MEMCPY(destAddr := ADR(typeClass), srcAddr := ADR(unknownCode), n := SIZEOF(typeClass));
narrowName := TOF_Core.SystemTypeClassConvertor.ToString(typeClass := typeClass);
wideName := TOF_Core.SystemTypeClassConvertor.ToWideString(typeClass := typeClass);
Assert.ThatBool(
	actual := narrowName = '4294967295',
	message := "STRING fallback must retain the unsigned code"
).IsTrue();
Assert.ThatBool(
	actual := wideName = "4294967295",
	message := "WSTRING fallback must retain the unsigned code"
).IsTrue();
END_METHOD

//! <summary>Borrows the concrete class name. Callers must not modify it.</summary>
{attribute 'monitoring' := 'call'}
PROPERTY ClassName : REFERENCE TO STRING
GET
ClassName REF= _ClassName;
END_GET
END_PROPERTY

//! <summary>Borrows the compiler-initialized namespace name. Callers must not modify it.</summary>
{attribute 'monitoring' := 'call'}
PROPERTY NamespaceName : REFERENCE TO STRING
GET
NamespaceName REF= CurrentNamespace.Name;
END_GET
END_PROPERTY

//! <summary>Reports the concrete instance size in bytes.</summary>
{attribute 'monitoring' := 'call'}
PROPERTY SelfSize : ULINT
GET
SelfSize := XSIZEOF(THIS^);
END_GET
END_PROPERTY

END_FUNCTION_BLOCK

// ---- Tests/Core/SystemTypeClassDiagnosticsTest.TcPOU
(*
SPDX-FileCopyrightText: c 2026 Oleksandr Tiutyk <trofimich@gmail.com>
SPDX-License-Identifier: MIT
License: https://opensource.org/license/mit
*)

(*!
<summary>Checks runtime type names in exceptions and unsupported-value diagnostics.</summary>
<description>
Uses run-local fixtures and references that are used only within the executing PLC task.
The runner binds assertions to the instance address. Keep the instance at that address for its run.
</description>
*)

{attribute 'no_assign'}
{attribute 'no_explicit_call' := 'do not call this function block directly'}
FUNCTION_BLOCK SystemTypeClassDiagnosticsTest EXTENDS TOF_Testing.SingleCycleTest
VAR_STAT
	{attribute 'hide'}
	_ClassName : STRING := __POUNAME();
END_VAR

(*!
<summary>Checks runtime names in public string rejection messages and unsupported-value markers.</summary>
<description>
Catches deliberate type errors to inspect the message while the task-owned exception is alive.
Checks the exception type and exact message. A failed append must preserve its target.
Unsupported arrays must retain a readable TYPE_ARRAY marker and size.
</description>
*)
METHOD PROTECTED ExecuteTest
VAR
	narrowTarget : STRING(10) := 'keep';
	wideTarget : WSTRING(10) := "keep";
	narrowMessage : STRING(255);
	wideMessage : WSTRING(255);
	unsupportedValue : ARRAY [0..0] OF DINT;
	exceptionCode : __SYSTEM.ExceptionCode;
	caughtException : TOF_Core.IException;
	notSupportedException : TOF_Core.INotSupportedException;
	message : TOF_Core.ERROR_MESSAGE;
END_VAR
// Capture the deliberate type error so its specific payload can be checked.
__TRY
	TOF_Core.WideStrings.AppendFit255(narrowTarget, "x");
__CATCH(exceptionCode)
	caughtException := TOF_Core.ExceptionManager.GetLastException(
		exceptionCode := exceptionCode,
		catchPointNamespaceName := NamespaceName,
		catchPointPOUName := __POUNAME(),
		catchPointPosition := __POSITION()
	);
__ENDTRY

IF __QUERYINTERFACE(caughtException, notSupportedException) THEN
	message := caughtException.GetMessage();
	Assert.ThatBool(
		actual := message = "Not supported type TYPE_STRING",
		message := "WideStrings.AppendFit255 must name TYPE_STRING in the exception message"
	).IsTrue();
ELSE
	RecordFailure(message := "WideStrings.AppendFit255 must reject TYPE_STRING with NotSupportedException");
END_IF

caughtException := 0;

// Capture the deliberate type error so its specific payload can be checked.
__TRY
	TOF_Core.Strings.AppendFit255(wideTarget, 'x');
__CATCH(exceptionCode)
	caughtException := TOF_Core.ExceptionManager.GetLastException(
		exceptionCode := exceptionCode,
		catchPointNamespaceName := NamespaceName,
		catchPointPOUName := __POUNAME(),
		catchPointPosition := __POSITION()
	);
__ENDTRY

IF __QUERYINTERFACE(caughtException, notSupportedException) THEN
	message := caughtException.GetMessage();
	Assert.ThatBool(
		actual := message = "Not supported type TYPE_WSTRING",
		message := "Strings.AppendFit255 must name TYPE_WSTRING in the exception message"
	).IsTrue();
ELSE
	RecordFailure(message := "Strings.AppendFit255 must reject TYPE_WSTRING with NotSupportedException");
END_IF

Assert.ThatBool(actual := narrowTarget = 'keep', message := "Rejected STRING target changed").IsTrue();
Assert.ThatBool(actual := wideTarget = "keep", message := "Rejected WSTRING target changed").IsTrue();

narrowMessage := TOF_Core.Strings.AnyToString255(value := unsupportedValue);
wideMessage := TOF_Core.WideStrings.AnyToString255(value := unsupportedValue);
Assert.ThatBool(
	actual := TOF_Core.Strings.Contains(stringToSearchIn := narrowMessage, stringToFind := 'type class: TYPE_ARRAY'),
	message := "STRING marker must identify the unsupported DINT array"
).IsTrue();
Assert.ThatBool(
	actual := TOF_Core.WideStrings.Contains(
		stringToSearchIn := wideMessage,
		stringToFind := "type class: TYPE_ARRAY"
	),
	message := "WSTRING marker must identify the unsupported DINT array"
).IsTrue();
Assert.ThatBool(
	actual := TOF_Core.Strings.Contains(stringToSearchIn := narrowMessage, stringToFind := 'size: 4 bytes'),
	message := "STRING marker must include the size of one DINT"
).IsTrue();
Assert.ThatBool(
	actual := TOF_Core.WideStrings.Contains(stringToSearchIn := wideMessage, stringToFind := "size: 4 bytes"),
	message := "WSTRING marker must include the size of one DINT"
).IsTrue();
END_METHOD

//! <summary>Borrows the concrete class name. Callers must not modify it.</summary>
{attribute 'monitoring' := 'call'}
PROPERTY ClassName : REFERENCE TO STRING
GET
ClassName REF= _ClassName;
END_GET
END_PROPERTY

//! <summary>Borrows the compiler-initialized namespace name. Callers must not modify it.</summary>
{attribute 'monitoring' := 'call'}
PROPERTY NamespaceName : REFERENCE TO STRING
GET
NamespaceName REF= CurrentNamespace.Name;
END_GET
END_PROPERTY

//! <summary>Reports the concrete instance size in bytes.</summary>
{attribute 'monitoring' := 'call'}
PROPERTY SelfSize : ULINT
GET
SelfSize := XSIZEOF(THIS^);
END_GET
END_PROPERTY

END_FUNCTION_BLOCK

// ---- Tests/Core/GenericBorrowedWritesTest.TcPOU
(*
SPDX-FileCopyrightText: c 2026 Oleksandr Tiutyk <trofimich@gmail.com>
SPDX-License-Identifier: MIT
License: https://opensource.org/license/mit
*)

(*!
<summary>Checks compatible writes and nonmutating rejection in borrowed storage.</summary>
<description>
Uses run-local fixtures and references that are used only within the executing PLC task.
The runner binds assertions to the instance address. Keep the instance at that address for its run.
</description>
*)

{attribute 'no_assign'}
{attribute 'no_explicit_call' := 'do not call this function block directly'}
FUNCTION_BLOCK GenericBorrowedWritesTest EXTENDS TOF_Testing.SingleCycleTest
VAR_STAT
	{attribute 'hide'}
	_ClassName : STRING := __POUNAME();
END_VAR

(*!
<summary>Checks compatible borrowed writes and direct rejection of type and capacity mismatches.</summary>
<description>
Both Try entry points exercise live source and destination storage. Each rejection preserves the destination
and the known task exception. The original string descriptor address is captured before writes. Borrowed
descriptors and their addresses stay within the callback.
</description>
*)
METHOD PROTECTED ExecuteTest
VAR
	destination : TOF_Core.GENERIC_VALUE;
	stored : REAL := 3.0;
	integerInput : DINT := 5;
	realInput : REAL := 5.0;
	shortDestination : TOF_Core.GENERIC_VALUE;
	originalShortAddress : POINTER TO BYTE;
	shortText : STRING(1) := 'x';
	longText : STRING(8) := 'longer';
	replacementText : STRING(1) := 'y';
	source : TOF_Core.GENERIC_VALUE;
	accepted : BOOL;
	exceptionCode : __SYSTEM.ExceptionCode;
	sentinel : TOF_Core.IException;
	afterFailure : TOF_Core.IException;
	sentinelMessage : TOF_Core.ERROR_MESSAGE := "Try write exception sentinel";
	standardException : TOF_Core.IStandardException;
END_VAR
// Establish a known task payload so a false result cannot hide a replaced exception.
__TRY
	TOF_Core.Exceptions.ThrowStandard(
		sourceNamespaceName := NamespaceName,
		sourceClassName := ClassName,
		sourcePOUName := __POUNAME(),
		sourcePosition := __POSITION(),
		message := sentinelMessage
	);
__CATCH(exceptionCode)
	sentinel := TOF_Core.ExceptionManager.GetLastException(
		exceptionCode := exceptionCode,
		catchPointNamespaceName := NamespaceName,
		catchPointPOUName := __POUNAME(),
		catchPointPosition := __POSITION()
	);
__ENDTRY

IF NOT __QUERYINTERFACE(sentinel, standardException) THEN
	RecordFailure(message := "The test must establish a standard exception before attempting writes");
	RETURN;
END_IF

Assert.ThatBool(
	actual := standardException.SourceMessage = sentinelMessage,
	message := "The task payload must be the test sentinel"
).IsTrue();

destination := TOF_Core.GenericValueFactory.FromRealReference(value := stored);
accepted := destination.TryChangeValueByAny(value := integerInput);
afterFailure := TOF_Core.ExceptionManager.GetLastException(
	exceptionCode := __SYSTEM.ExceptionCode.RTSEXCPT_USER_EXCEPTION_BASE,
	catchPointNamespaceName := NamespaceName,
	catchPointPOUName := __POUNAME(),
	catchPointPosition := __POSITION()
);
Assert.ThatBool(actual := accepted, message := "DINT cannot replace REAL storage").IsFalse();
Assert.ThatBool(actual := sentinel = afterFailure, message := "Type rejection must preserve the task payload").IsTrue();
Assert.ThatReal(actual := stored, message := "Rejected DINT changed REAL storage").ToBe(expected := REAL#3.0);

shortDestination := TOF_Core.GenericValueFactory.FromAny(
	value := shortText,
	isObject := FALSE,
	memoryManagementBehavior := TOF_Core.GENERIC_MEMORY_MANAGEMENT_BEHAVIOR.STORE_ORIGINAL_REFERENCE_AND_NOT_OWNS_MEMORY
);
originalShortAddress := shortDestination.Address;
source := TOF_Core.GenericValueFactory.FromAny(
	value := longText,
	isObject := FALSE,
	memoryManagementBehavior := TOF_Core.GENERIC_MEMORY_MANAGEMENT_BEHAVIOR.STORE_ORIGINAL_REFERENCE_AND_NOT_OWNS_MEMORY
);
accepted := shortDestination.TryChangeValueByAnyType(value := source.AsAnyType());
afterFailure := TOF_Core.ExceptionManager.GetLastException(
	exceptionCode := __SYSTEM.ExceptionCode.RTSEXCPT_USER_EXCEPTION_BASE,
	catchPointNamespaceName := NamespaceName,
	catchPointPOUName := __POUNAME(),
	catchPointPosition := __POSITION()
);
Assert.ThatBool(actual := accepted, message := "Undersized storage must reject the string copy").IsFalse();
Assert.ThatBool(
	actual := sentinel = afterFailure,
	message := "Capacity rejection must preserve the task payload"
).IsTrue();
Assert.ThatBool(
	actual := standardException.SourceMessage = sentinelMessage,
	message := "Type and capacity rejections must preserve the original exception text"
).IsTrue();
Assert.ThatBool(actual := shortText = 'x', message := "Rejected size changed STRING storage").IsTrue();

accepted := destination.TryChangeValueByAny(value := realInput);
Assert.ThatBool(actual := accepted, message := "Compatible REAL storage must accept a copy").IsTrue();
Assert.ThatReal(actual := stored, message := "Compatible REAL copy lost the value").ToBe(expected := realInput);

source := TOF_Core.GenericValueFactory.FromAny(
	value := replacementText,
	isObject := FALSE,
	memoryManagementBehavior := TOF_Core.GENERIC_MEMORY_MANAGEMENT_BEHAVIOR.STORE_ORIGINAL_REFERENCE_AND_NOT_OWNS_MEMORY
);
accepted := shortDestination.TryChangeValueByAnyType(value := source.AsAnyType());
Assert.ThatBool(actual := accepted, message := "Equal STRING capacity must accept a copy").IsTrue();
Assert.ThatBool(actual := shortText = 'y', message := "Compatible STRING copy lost the value").IsTrue();
Assert.ThatBool(
	actual := shortDestination.Address = originalShortAddress
		AND_THEN shortDestination.Size = XSIZEOF(shortText)
		AND_THEN shortDestination.TypeClass = TOF_Core.GENERIC_TYPE_CLASS.STRING_8
		AND_THEN NOT shortDestination.IsMemoryOwner,
	message := "STRING writes must preserve size, type, address and borrowed ownership"
).IsTrue();
END_METHOD

//! <summary>Borrows the concrete class name. Callers must not modify it.</summary>
{attribute 'monitoring' := 'call'}
PROPERTY ClassName : REFERENCE TO STRING
GET
ClassName REF= _ClassName;
END_GET
END_PROPERTY

//! <summary>Borrows the compiler-initialized namespace name. Callers must not modify it.</summary>
{attribute 'monitoring' := 'call'}
PROPERTY NamespaceName : REFERENCE TO STRING
GET
NamespaceName REF= CurrentNamespace.Name;
END_GET
END_PROPERTY

//! <summary>Reports the concrete instance size in bytes.</summary>
{attribute 'monitoring' := 'call'}
PROPERTY SelfSize : ULINT
GET
SelfSize := XSIZEOF(THIS^);
END_GET
END_PROPERTY

END_FUNCTION_BLOCK

// ---- Tests/Core/RandomTestGroup.TcPOU
(*
SPDX-FileCopyrightText: c 2026 Oleksandr Tiutyk <trofimich@gmail.com>
SPDX-License-Identifier: MIT
License: https://opensource.org/license/mit
*)

(*!
<summary>Groups random range and dispersion contracts.</summary>
<description>
Owns the independent child instances and their fixed registration array. Use from one PLC task at a stable address.
</description>
*)

{attribute 'no_assign'}
{attribute 'no_explicit_call' := 'do not call this function block directly'}
FUNCTION_BLOCK RandomTestGroup EXTENDS TOF_Testing.TestGroup<3>
VAR_STAT
	{attribute 'hide'}
	_ClassName : STRING := __POUNAME();
END_VAR
VAR
	_Range : RandomRangeTest(name := "GetInRange", parent := THIS^);
	_AbsoluteDispersion : RandomAbsoluteDispersionTest(name := "GetWithDispersion", parent := THIS^);
	_PercentageDispersion : RandomPercentageDispersionTest(name := "GetWithDispersionPercent", parent := THIS^);

	_Children : ARRAY [0.._ChildCount - 1] OF TOF_Testing.ITestElement :=
	[
		_Range,
		_AbsoluteDispersion,
		_PercentageDispersion
	];
END_VAR

//! <summary>Borrows the fixed child array. Callers must not modify it.</summary>
{attribute 'monitoring' := 'call'}
PROPERTY Children : REFERENCE TO ARRAY [0.._ChildCount - 1] OF TOF_Testing.ITestElement
GET
Children REF= _Children;
END_GET
END_PROPERTY

//! <summary>Borrows the concrete class name. Callers must not modify it.</summary>
{attribute 'monitoring' := 'call'}
PROPERTY ClassName : REFERENCE TO STRING
GET
ClassName REF= _ClassName;
END_GET
END_PROPERTY

//! <summary>Borrows the compiler-initialized namespace name. Callers must not modify it.</summary>
{attribute 'monitoring' := 'call'}
PROPERTY NamespaceName : REFERENCE TO STRING
GET
NamespaceName REF= CurrentNamespace.Name;
END_GET
END_PROPERTY

//! <summary>Reports the concrete instance size in bytes.</summary>
{attribute 'monitoring' := 'call'}
PROPERTY SelfSize : ULINT
GET
SelfSize := XSIZEOF(THIS^);
END_GET
END_PROPERTY

END_FUNCTION_BLOCK

// ---- Tests/Core/RandomRangeTest.TcPOU
(*
SPDX-FileCopyrightText: c 2026 Oleksandr Tiutyk <trofimich@gmail.com>
SPDX-License-Identifier: MIT
License: https://opensource.org/license/mit
*)

(*!
<summary>Checks random scaling and a single-point interval.</summary>
<description>
Owns a generator used by one PLC task. Each run checks the same bounds against fresh samples.
The runner binds assertions to the instance address. Keep the instance at that address for its run.
</description>
*)

{attribute 'no_assign'}
{attribute 'no_explicit_call' := 'do not call this function block directly'}
FUNCTION_BLOCK RandomRangeTest EXTENDS TOF_Testing.SingleCycleTest
VAR_STAT
	{attribute 'hide'}
	_ClassName : STRING := __POUNAME();
END_VAR
VAR
	_Random : TOF_Core.Random;
END_VAR

//! <summary>Checks a single-point range and samples an inclusive interval.</summary>
METHOD PROTECTED ExecuteTest
VAR
	value : LREAL;
	i : INT;
END_VAR
value := _Random.GetInRange(minValue := LREAL#-7.5, maxValue := LREAL#-7.5);
Assert.ThatLongReal(
	actual := value,
	message := "A single-point range must return its bound"
).ToBe(expected := LREAL#-7.5);

FOR i := 1 TO 21 DO
	value := _Random.GetInRange(minValue := LREAL#100.0, maxValue := LREAL#200.0);
	Assert.ThatLongReal(
		actual := value,
		message := "GetInRange sample below 100"
	).IsGreaterThanOrEquals(expected := LREAL#100.0);
	Assert.ThatLongReal(
		actual := value,
		message := "GetInRange sample above 200"
	).IsLessThanOrEquals(expected := LREAL#200.0);
END_FOR
END_METHOD

//! <summary>Borrows the concrete class name. Callers must not modify it.</summary>
{attribute 'monitoring' := 'call'}
PROPERTY ClassName : REFERENCE TO STRING
GET
ClassName REF= _ClassName;
END_GET
END_PROPERTY

//! <summary>Borrows the compiler-initialized namespace name. Callers must not modify it.</summary>
{attribute 'monitoring' := 'call'}
PROPERTY NamespaceName : REFERENCE TO STRING
GET
NamespaceName REF= CurrentNamespace.Name;
END_GET
END_PROPERTY

//! <summary>Reports the concrete instance size in bytes.</summary>
{attribute 'monitoring' := 'call'}
PROPERTY SelfSize : ULINT
GET
SelfSize := XSIZEOF(THIS^);
END_GET
END_PROPERTY

END_FUNCTION_BLOCK

// ---- Tests/Core/RandomAbsoluteDispersionTest.TcPOU
(*
SPDX-FileCopyrightText: c 2026 Oleksandr Tiutyk <trofimich@gmail.com>
SPDX-License-Identifier: MIT
License: https://opensource.org/license/mit
*)

(*!
<summary>Checks absolute dispersion and independent output clamps.</summary>
<description>
Owns a generator used by one PLC task. Each run checks the same bounds against fresh samples.
The runner binds assertions to the instance address. Keep the instance at that address for its run.
</description>
*)

{attribute 'no_assign'}
{attribute 'no_explicit_call' := 'do not call this function block directly'}
FUNCTION_BLOCK RandomAbsoluteDispersionTest EXTENDS TOF_Testing.SingleCycleTest
VAR_STAT
	{attribute 'hide'}
	_ClassName : STRING := __POUNAME();
END_VAR
VAR
	_Random : TOF_Core.Random;
END_VAR

//! <summary>Checks zero dispersion and bounds that must clamp independently of the generated sample.</summary>
METHOD PROTECTED ExecuteTest
VAR
	value : LREAL;
	i : INT;
END_VAR
value := _Random.GetWithDispersion(baseValue := LREAL#12.5, dispersion := LREAL#0.0);
Assert.ThatLongReal(actual := value, message := "Zero dispersion must return the base").ToBe(expected := LREAL#12.5);

value := _Random.GetWithDispersion(baseValue := LREAL#100.0, dispersion := LREAL#10.0, minValue := LREAL#120.0);
Assert.ThatLongReal(
	actual := value,
	message := "Lower bound alone must clamp any sample"
).ToBe(expected := LREAL#120.0);

value := _Random.GetWithDispersion(baseValue := LREAL#100.0, dispersion := LREAL#10.0, maxValue := LREAL#80.0);
Assert.ThatLongReal(actual := value, message := "Upper bound alone must clamp any sample").ToBe(expected := LREAL#80.0);

FOR i := 1 TO 21 DO
	value := _Random.GetWithDispersion(baseValue := LREAL#100.0, dispersion := LREAL#10.0);
	Assert.ThatLongReal(
	actual := value,
	message := "Absolute dispersion sample below 90"
).IsGreaterThanOrEquals(
		expected := LREAL#90.0
	);
	Assert.ThatLongReal(
	actual := value,
	message := "Absolute dispersion sample above 110"
).IsLessThanOrEquals(
		expected := LREAL#110.0
	);
END_FOR
END_METHOD

//! <summary>Borrows the concrete class name. Callers must not modify it.</summary>
{attribute 'monitoring' := 'call'}
PROPERTY ClassName : REFERENCE TO STRING
GET
ClassName REF= _ClassName;
END_GET
END_PROPERTY

//! <summary>Borrows the compiler-initialized namespace name. Callers must not modify it.</summary>
{attribute 'monitoring' := 'call'}
PROPERTY NamespaceName : REFERENCE TO STRING
GET
NamespaceName REF= CurrentNamespace.Name;
END_GET
END_PROPERTY

//! <summary>Reports the concrete instance size in bytes.</summary>
{attribute 'monitoring' := 'call'}
PROPERTY SelfSize : ULINT
GET
SelfSize := XSIZEOF(THIS^);
END_GET
END_PROPERTY

END_FUNCTION_BLOCK

// ---- Tests/Core/RandomPercentageDispersionTest.TcPOU
(*
SPDX-FileCopyrightText: c 2026 Oleksandr Tiutyk <trofimich@gmail.com>
SPDX-License-Identifier: MIT
License: https://opensource.org/license/mit
*)

